   1:  PR[91,3] = PR[90,3] + 75.576;
   1:L PR[91] R[100]mm/sec CNT100;
   1:  PR[91,1] = PR[90,1] + -58.214;
   1:  PR[91,2] = PR[90,2] + 18.783;
   1:  PR[91,3] = PR[90,3] + 75.587;
   1:L PR[91] R[100]mm/sec CNT100;
   1:  PR[91] = PR[90];
   1:  PR[91,1] = PR[90,1] + -61.321;
   1:  PR[91,2] = PR[90,2] + 16.488;
   1:  PR[91,3] = PR[90,3] + 76.895;
   1:L PR[91] R[100]mm/sec CNT100;
   1:  PR[91,1] = PR[90,1] + -61.751;
   1:  PR[91,2] = PR[90,2] + 16.148;
   1:  PR[91,3] = PR[90,3] + 75.611;
   1:L PR[91] R[100]mm/sec CNT100;
   1:  PR[91,1] = PR[90,1] + -63.245;
   1:  PR[91,2] = PR[90,2] + 14.908;
   1:  PR[91,3] = PR[90,3] + 75.613;
   1:L PR[91] R[100]mm/sec CNT100;
   1:  PR[91,1] = PR[90,1] + -65.760;
   1:  PR[91,2] = PR[90,2] + 12.618;
   1:  PR[91,3] = PR[90,3] + 75.621;
   1:L PR[91] R[100]mm/sec CNT100;
   1:  PR[91,1] = PR[90,1] + -68.800;
   1:  PR[91,2] = PR[90,2] + 8.357;
   1:  PR[91,3] = PR[90,3] + 75.634;
   1:L PR[91] R[100]mm/sec CNT100;
   1:  PR[91,1] = PR[90,1] + -70.612;
   1:  PR[91,2] = PR[90,2] + 3.865;
   1:  PR[91,3] = PR[90,3] + 75.654;
   1:L PR[91] R[100]mm/sec CNT100;
   1:  PR[91,1] = PR[90,1] + -70.919;
   1:  PR[91,2] = PR[90,2] + 1.527;
   1:  PR[91,3] = PR[90,3] + 75.672;
   1:L PR[91] R[100]mm/sec CNT100;
   1:  PR[91,1] = PR[90,1] + -71.311;
   1:  PR[91,2] = PR[90,2] + -0.699;
   1:  PR[91,3] = PR[90,3] + 75.682;
   1:L PR[91] R[100]mm/sec CNT100;
   1:  PR[91,1] = PR[90,1] + -71.180;
   1:  PR[91,2] = PR[90,2] + -1.329;
   1:  PR[91,3] = PR[90,3] + 75.690;
   1:L PR[91] R[100]mm/sec CNT100;
   1:  PR[91,1] = PR[90,1] + -70.648;
   1:  PR[91,2] = PR[90,2] + -5.468;
   1:  PR[91,3] = PR[90,3] + 75.693;
   1:L PR[91] R[100]mm/sec CNT100;
   1:  PR[91,1] = PR[90,1] + -68.806;
   1:  PR[91,2] = PR[90,2] + -10.057;
   1:  PR[91,3] = PR[90,3] + 75.709;
   1:L PR[91] R[100]mm/sec CNT100;
   1:  PR[91,1] = PR[90,1] + -68.274;
   1:  PR[91,2] = PR[90,2] + -10.806;
   1:  PR[91,3] = PR[90,3] + 75.728;
   1:L PR[91] R[100]mm/sec CNT100;
   1:  PR[91,1] = PR[90,1] + -65.619;
   1:  PR[91,2] = PR[90,2] + -14.212;
   1:  PR[91,3] = PR[90,3] + 75.731;
   1:L PR[91] R[100]mm/sec CNT100;
   1:  PR[91,1] = PR[90,1] + -64.867;
   1:  PR[91,2] = PR[90,2] + -14.891;
   1:  PR[91,3] = PR[90,3] + 75.748;
   1:L PR[91] R[100]mm/sec CNT100;
   1:  PR[91,1] = PR[90,1] + -61.355;
   1:  PR[91,2] = PR[90,2] + -17.818;
   1:  PR[91,3] = PR[90,3] + 75.752;
   1:L PR[91] R[100]mm/sec CNT100;
   1:  PR[91,1] = PR[90,1] + -58.279;
   1:  PR[91,2] = PR[90,2] + -19.704;
   1:  PR[91,3] = PR[90,3] + 75.769;
   1:L PR[91] R[100]mm/sec CNT100;
   1:  PR[91,1] = PR[90,1] + -56.388;
   1:  PR[91,2] = PR[90,2] + -20.757;
   1:  PR[91,3] = PR[90,3] + 75.783;
   1:L PR[91] R[100]mm/sec CNT100;
   1:  PR[91,1] = PR[90,1] + -52.808;
   1:  PR[91,2] = PR[90,2] + -22.216;
   1:  PR[91,3] = PR[90,3] + 75.791;
   1:L PR[91] R[100]mm/sec CNT100;
   1:  PR[91,1] = PR[90,1] + -51.042;
   1:  PR[91,2] = PR[90,2] + -22.876;
   1:  PR[91,3] = PR[90,3] + 75.806;
   1:L PR[91] R[100]mm/sec CNT100;
   1:  PR[91,1] = PR[90,1] + -50.028;
   1:  PR[91,2] = PR[90,2] + -23.222;
   1:  PR[91,3] = PR[90,3] + 75.813;
   1:L PR[91] R[100]mm/sec CNT100;
   1:  PR[91,1] = PR[90,1] + -45.759;
   1:  PR[91,2] = PR[90,2] + -24.206;
   1:  PR[91,3] = PR[90,3] + 75.817;
   1:L PR[91] R[100]mm/sec CNT100;
   1:  PR[91,1] = PR[90,1] + -40.300;
   1:  PR[91,2] = PR[90,2] + -25.279;
   1:  PR[91,3] = PR[90,3] + 75.834;
   1:L PR[91] R[100]mm/sec CNT100;
   1:  PR[91,1] = PR[90,1] + -33.010;
   1:  PR[91,2] = PR[90,2] + -25.861;
   1:  PR[91,3] = PR[90,3] + 75.855;
   1:L PR[91] R[100]mm/sec CNT100;
   1:  PR[91,1] = PR[90,1] + -26.617;
   1:  PR[91,2] = PR[90,2] + -26.061;
   1:  PR[91,3] = PR[90,3] + 75.884;
   1:L PR[91] R[100]mm/sec CNT100;
   1:  PR[91,1] = PR[90,1] + -16.860;
   1:  PR[91,2] = PR[90,2] + -25.700;
   1:  PR[91,3] = PR[90,3] + 75.908;
   1:L PR[91] R[100]mm/sec CNT100;
   1:  PR[91,1] = PR[90,1] + -16.514;
   1:  PR[91,2] = PR[90,2] + -25.675;
   1:  PR[91,3] = PR[90,3] + 75.945;
   1:L PR[91] R[100]mm/sec CNT100;
   1:  PR[91,1] = PR[90,1] + -11.759;
   1:  PR[91,2] = PR[90,2] + -25.135;
   1:  PR[91,3] = PR[90,3] + 75.947;
   1:L PR[91] R[100]mm/sec CNT100;
   1:  PR[91,1] = PR[90,1] + -10.834;
   1:  PR[91,2] = PR[90,2] + -25.105;
   1:  PR[91,3] = PR[90,3] + 75.965;
   1:L PR[91] R[100]mm/sec CNT100;
   1:  PR[91,1] = PR[90,1] + -9.602;
   1:  PR[91,2] = PR[90,2] + -24.937;
   1:  PR[91,3] = PR[90,3] + 75.969;
   1:L PR[91] R[100]mm/sec CNT100;
   1:  PR[91,1] = PR[90,1] + -7.923;
   1:  PR[91,2] = PR[90,2] + -25.330;
   1:  PR[91,3] = PR[90,3] + 75.973;
   1:L PR[91] R[100]mm/sec CNT100;
   1:  PR[91,1] = PR[90,1] + -3.823;
   1:  PR[91,2] = PR[90,2] + -25.725;
   1:  PR[91,3] = PR[90,3] + 75.980;
   1:L PR[91] R[100]mm/sec CNT100;
   1:  PR[91,1] = PR[90,1] + -1.693;
   1:  PR[91,2] = PR[90,2] + -25.951;
   1:  PR[91,3] = PR[90,3] + 75.996;
   1:L PR[91] R[100]mm/sec CNT100;
   1:  PR[91,1] = PR[90,1] + -0.935;
   1:  PR[91,2] = PR[90,2] + -25.962;
   1:  PR[91,3] = PR[90,3] + 76.004;
   1:L PR[91] R[100]mm/sec CNT100;
   1:  PR[91,1] = PR[90,1] + 4.101;
   1:  PR[91,2] = PR[90,2] + -25.614;
   1:  PR[91,3] = PR[90,3] + 76.007;
   1:L PR[91] R[100]mm/sec CNT100;
   1:  PR[91,1] = PR[90,1] + 6.267;
   1:  PR[91,2] = PR[90,2] + -25.357;
   1:  PR[91,3] = PR[90,3] + 76.026;
   1:L PR[91] R[100]mm/sec CNT100;
   1:  PR[91,1] = PR[90,1] + 6.639;
   1:  PR[91,2] = PR[90,2] + -25.282;
   1:  PR[91,3] = PR[90,3] + 76.035;
   1:L PR[91] R[100]mm/sec CNT100;
   1:  PR[91,1] = PR[90,1] + 9.233;
   1:  PR[91,2] = PR[90,2] + -24.616;
   1:  PR[91,3] = PR[90,3] + 76.036;
   1:L PR[91] R[100]mm/sec CNT100;
   1:  PR[91,1] = PR[90,1] + 10.669;
   1:  PR[91,2] = PR[90,2] + -25.276;
   1:  PR[91,3] = PR[90,3] + 76.046;
   1:L PR[91] R[100]mm/sec CNT100;
   1:  PR[91,1] = PR[90,1] + 11.562;
   1:  PR[91,2] = PR[90,2] + -25.519;
   1:  PR[91,3] = PR[90,3] + 76.052;
   1:L PR[91] R[100]mm/sec CNT100;
   1:  PR[91,1] = PR[90,1] + 16.871;
   1:  PR[91,2] = PR[90,2] + -26.664;
   1:  PR[91,3] = PR[90,3] + 76.056;
   1:L PR[91] R[100]mm/sec CNT100;
   1:  PR[91,1] = PR[90,1] + 18.179;
   1:  PR[91,2] = PR[90,2] + -26.717;
   1:  PR[91,3] = PR[90,3] + 76.077;
   1:L PR[91] R[100]mm/sec CNT100;
   1:  PR[91,1] = PR[90,1] + 23.121;
   1:  PR[91,2] = PR[90,2] + -26.558;
   1:  PR[91,3] = PR[90,3] + 76.082;
   1:L PR[91] R[100]mm/sec CNT100;
   1:  PR[91,1] = PR[90,1] + 25.230;
   1:  PR[91,2] = PR[90,2] + -26.240;
   1:  PR[91,3] = PR[90,3] + 76.101;
   1:L PR[91] R[100]mm/sec CNT100;
   1:  PR[91,1] = PR[90,1] + 28.911;
   1:  PR[91,2] = PR[90,2] + -27.201;
   1:  PR[91,3] = PR[90,3] + 76.109;
   1:L PR[91] R[100]mm/sec CNT100;
   1:  PR[91,1] = PR[90,1] + 30.544;
   1:  PR[91,2] = PR[90,2] + -27.575;
   1:  PR[91,3] = PR[90,3] + 76.124;
   1:L PR[91] R[100]mm/sec CNT100;
   1:  PR[91,1] = PR[90,1] + 35.732;
   1:  PR[91,2] = PR[90,2] + -27.991;
   1:  PR[91,3] = PR[90,3] + 76.130;
   1:L PR[91] R[100]mm/sec CNT100;
   1:  PR[91,1] = PR[90,1] + 36.008;
   1:  PR[91,2] = PR[90,2] + -27.986;
   1:  PR[91,3] = PR[90,3] + 76.150;
   1:L PR[91] R[100]mm/sec CNT100;
   1:  PR[91,1] = PR[90,1] + 40.601;
   1:  PR[91,2] = PR[90,2] + -27.632;
   1:  PR[91,3] = PR[90,3] + 76.151;
   1:L PR[91] R[100]mm/sec CNT100;
   1:  PR[91,1] = PR[90,1] + 43.395;
   1:  PR[91,2] = PR[90,2] + -27.151;
   1:  PR[91,3] = PR[90,3] + 76.169;
   1:L PR[91] R[100]mm/sec CNT100;
   1:  PR[91,1] = PR[90,1] + 44.903;
   1:  PR[91,2] = PR[90,2] + -26.790;
   1:  PR[91,3] = PR[90,3] + 76.180;
   1:L PR[91] R[100]mm/sec CNT100;
   1:  PR[91,1] = PR[90,1] + 47.079;
   1:  PR[91,2] = PR[90,2] + -26.059;
   1:  PR[91,3] = PR[90,3] + 76.186;
   1:L PR[91] R[100]mm/sec CNT100;
   1:  PR[91,1] = PR[90,1] + 49.432;
   1:  PR[91,2] = PR[90,2] + -25.424;
   1:  PR[91,3] = PR[90,3] + 76.194;
   1:L PR[91] R[100]mm/sec CNT100;
   1:  PR[91,1] = PR[90,1] + 51.453;
   1:  PR[91,2] = PR[90,2] + -24.639;
   1:  PR[91,3] = PR[90,3] + 76.204;
   1:L PR[91] R[100]mm/sec CNT100;
   1:  PR[91,1] = PR[90,1] + 53.638;
   1:  PR[91,2] = PR[90,2] + -23.715;
   1:  PR[91,3] = PR[90,3] + 76.212;
   1:L PR[91] R[100]mm/sec CNT100;
   1:  PR[91,1] = PR[90,1] + 55.403;
   1:  PR[91,2] = PR[90,2] + -22.742;
   1:  PR[91,3] = PR[90,3] + 76.221;
   1:L PR[91] R[100]mm/sec CNT100;
   1:  PR[91,1] = PR[90,1] + 57.643;
   1:  PR[91,2] = PR[90,2] + -21.692;
   1:  PR[91,3] = PR[90,3] + 76.229;
   1:L PR[91] R[100]mm/sec CNT100;
   1:  PR[91,1] = PR[90,1] + 61.600;
   1:  PR[91,2] = PR[90,2] + -19.230;
   1:  PR[91,3] = PR[90,3] + 76.238;
   1:L PR[91] R[100]mm/sec CNT100;
   1:  PR[91,1] = PR[90,1] + 65.239;
   1:  PR[91,2] = PR[90,2] + -16.034;
   1:  PR[91,3] = PR[90,3] + 76.256;
   1:L PR[91] R[100]mm/sec CNT100;
   1:  PR[91,1] = PR[90,1] + 66.422;
   1:  PR[91,2] = PR[90,2] + -14.530;
   1:  PR[91,3] = PR[90,3] + 76.275;
   1:L PR[91] R[100]mm/sec CNT100;
   1:  PR[91,1] = PR[90,1] + 68.582;
   1:  PR[91,2] = PR[90,2] + -11.849;
   1:  PR[91,3] = PR[90,3] + 76.282;
   1:L PR[91] R[100]mm/sec CNT100;
   1:  PR[91,1] = PR[90,1] + 69.577;
   1:  PR[91,2] = PR[90,2] + -10.060;
   1:  PR[91,3] = PR[90,3] + 76.295;
   1:L PR[91] R[100]mm/sec CNT100;
   1:  PR[91,1] = PR[90,1] + 70.915;
   1:  PR[91,2] = PR[90,2] + -7.005;
   1:  PR[91,3] = PR[90,3] + 76.303;
   1:L PR[91] R[100]mm/sec CNT100;
   1:  PR[91,1] = PR[90,1] + 71.354;
   1:  PR[91,2] = PR[90,2] + -5.640;
   1:  PR[91,3] = PR[90,3] + 76.316;
   1:L PR[91] R[100]mm/sec CNT100;
   1:  PR[91,1] = PR[90,1] + 71.890;
   1:  PR[91,2] = PR[90,2] + -1.894;
   1:  PR[91,3] = PR[90,3] + 76.321;
   1:L PR[91] R[100]mm/sec CNT100;
   1:  PR[91,1] = PR[90,1] + 72.009;
   1:  PR[91,2] = PR[90,2] + -0.768;
   1:  PR[91,3] = PR[90,3] + 76.336;
   1:L PR[91] R[100]mm/sec CNT100;
   1:  PR[91,1] = PR[90,1] + 71.482;
   1:  PR[91,2] = PR[90,2] + 2.880;
   1:  PR[91,3] = PR[90,3] + 76.340;
   1:L PR[91] R[100]mm/sec CNT100;
   1:  PR[91,1] = PR[90,1] + 71.343;
   1:  PR[91,2] = PR[90,2] + 4.216;
   1:  PR[91,3] = PR[90,3] + 76.354;
   1:L PR[91] R[100]mm/sec CNT100;
   1:  PR[91,1] = PR[90,1] + 70.915;
   1:  PR[91,2] = PR[90,2] + 5.544;
   1:  PR[91,3] = PR[90,3] + 76.359;
   1:L PR[91] R[100]mm/sec CNT100;
   1:  PR[91,1] = PR[90,1] + 69.579;
   1:  PR[91,2] = PR[90,2] + 8.598;
   1:  PR[91,3] = PR[90,3] + 76.365;
   1:L PR[91] R[100]mm/sec CNT100;
   1:  PR[91,1] = PR[90,1] + 68.577;
   1:  PR[91,2] = PR[90,2] + 10.401;
   1:  PR[91,3] = PR[90,3] + 76.378;
   1:L PR[91] R[100]mm/sec CNT100;
   1:  PR[91,1] = PR[90,1] + 67.100;
   1:  PR[91,2] = PR[90,2] + 12.290;
   1:  PR[91,3] = PR[90,3] + 76.386;
   1:L PR[91] R[100]mm/sec CNT100;
   1:  PR[91,1] = PR[90,1] + 65.254;
   1:  PR[91,2] = PR[90,2] + 14.562;
   1:  PR[91,3] = PR[90,3] + 76.395;
   1:L PR[91] R[100]mm/sec CNT100;
   1:  PR[91,1] = PR[90,1] + 61.600;
   1:  PR[91,2] = PR[90,2] + 17.771;
   1:  PR[91,3] = PR[90,3] + 76.406;
   1:L PR[91] R[100]mm/sec CNT100;
   1:  PR[91,1] = PR[90,1] + 57.643;
   1:  PR[91,2] = PR[90,2] + 20.234;
   1:  PR[91,3] = PR[90,3] + 76.425;
   1:L PR[91] R[100]mm/sec CNT100;
   1:  PR[91,1] = PR[90,1] + 55.403;
   1:  PR[91,2] = PR[90,2] + 21.284;
   1:  PR[91,3] = PR[90,3] + 76.442;
   1:L PR[91] R[100]mm/sec CNT100;
   1:  PR[91,1] = PR[90,1] + 53.638;
   1:  PR[91,2] = PR[90,2] + 22.256;
   1:  PR[91,3] = PR[90,3] + 76.452;
   1:L PR[91] R[100]mm/sec CNT100;
   1:  PR[91,1] = PR[90,1] + 51.453;
   1:  PR[91,2] = PR[90,2] + 23.180;
   1:  PR[91,3] = PR[90,3] + 76.460;
   1:L PR[91] R[100]mm/sec CNT100;
   1:  PR[91,1] = PR[90,1] + 49.432;
   1:  PR[91,2] = PR[90,2] + 23.965;
   1:  PR[91,3] = PR[90,3] + 76.469;
   1:L PR[91] R[100]mm/sec CNT100;
   1:  PR[91,1] = PR[90,1] + 47.079;
   1:  PR[91,2] = PR[90,2] + 24.601;
   1:  PR[91,3] = PR[90,3] + 76.477;
   1:L PR[91] R[100]mm/sec CNT100;
   1:  PR[91,1] = PR[90,1] + 44.903;
   1:  PR[91,2] = PR[90,2] + 25.331;
   1:  PR[91,3] = PR[90,3] + 76.486;
   1:L PR[91] R[100]mm/sec CNT100;
   1:  PR[91,1] = PR[90,1] + 43.395;
   1:  PR[91,2] = PR[90,2] + 25.692;
   1:  PR[91,3] = PR[90,3] + 76.495;
   1:L PR[91] R[100]mm/sec CNT100;
   1:  PR[91,1] = PR[90,1] + 40.601;
   1:  PR[91,2] = PR[90,2] + 26.173;
   1:  PR[91,3] = PR[90,3] + 76.501;
   1:L PR[91] R[100]mm/sec CNT100;
   1:  PR[91,1] = PR[90,1] + 36.008;
   1:  PR[91,2] = PR[90,2] + 26.528;
   1:  PR[91,3] = PR[90,3] + 76.512;
   1:L PR[91] R[100]mm/sec CNT100;
   1:  PR[91,1] = PR[90,1] + 35.732;
   1:  PR[91,2] = PR[90,2] + 26.532;
   1:  PR[91,3] = PR[90,3] + 76.530;
   1:L PR[91] R[100]mm/sec CNT100;
   1:  PR[91,1] = PR[90,1] + 30.544;
   1:  PR[91,2] = PR[90,2] + 26.116;
   1:  PR[91,3] = PR[90,3] + 76.531;
   1:L PR[91] R[100]mm/sec CNT100;
   1:  PR[91,1] = PR[90,1] + 28.911;
   1:  PR[91,2] = PR[90,2] + 25.742;
   1:  PR[91,3] = PR[90,3] + 76.551;
   1:L PR[91] R[100]mm/sec CNT100;
   1:  PR[91,1] = PR[90,1] + 25.230;
   1:  PR[91,2] = PR[90,2] + 24.781;
   1:  PR[91,3] = PR[90,3] + 76.557;
   1:L PR[91] R[100]mm/sec CNT100;
   1:  PR[91,1] = PR[90,1] + 23.121;
   1:  PR[91,2] = PR[90,2] + 25.099;
   1:  PR[91,3] = PR[90,3] + 76.572;
   1:L PR[91] R[100]mm/sec CNT100;
   1:  PR[91,1] = PR[90,1] + 18.179;
   1:  PR[91,2] = PR[90,2] + 25.258;
   1:  PR[91,3] = PR[90,3] + 76.580;
   1:L PR[91] R[100]mm/sec CNT100;
   1:  PR[91,1] = PR[90,1] + 16.870;
   1:  PR[91,2] = PR[90,2] + 25.205;
   1:  PR[91,3] = PR[90,3] + 76.599;
   1:L PR[91] R[100]mm/sec CNT100;
   1:  PR[91,1] = PR[90,1] + 11.562;
   1:  PR[91,2] = PR[90,2] + 24.060;
   1:  PR[91,3] = PR[90,3] + 76.604;
   1:L PR[91] R[100]mm/sec CNT100;
   1:  PR[91,1] = PR[90,1] + 10.668;
   1:  PR[91,2] = PR[90,2] + 23.817;
   1:  PR[91,3] = PR[90,3] + 76.625;
   1:L PR[91] R[100]mm/sec CNT100;
   1:  PR[91,1] = PR[90,1] + 9.232;
   1:  PR[91,2] = PR[90,2] + 23.158;
   1:  PR[91,3] = PR[90,3] + 76.628;
   1:L PR[91] R[100]mm/sec CNT100;
   1:  PR[91,1] = PR[90,1] + 6.658;
   1:  PR[91,2] = PR[90,2] + 23.820;
   1:  PR[91,3] = PR[90,3] + 76.634;
   1:L PR[91] R[100]mm/sec CNT100;
   1:  PR[91,1] = PR[90,1] + 6.292;
   1:  PR[91,2] = PR[90,2] + 23.894;
   1:  PR[91,3] = PR[90,3] + 76.644;
   1:L PR[91] R[100]mm/sec CNT100;
   1:  PR[91,1] = PR[90,1] + 4.125;
   1:  PR[91,2] = PR[90,2] + 24.151;
   1:  PR[91,3] = PR[90,3] + 76.646;
   1:L PR[91] R[100]mm/sec CNT100;
   1:  PR[91,1] = PR[90,1] + -0.919;
   1:  PR[91,2] = PR[90,2] + 24.504;
   1:  PR[91,3] = PR[90,3] + 76.654;
   1:L PR[91] R[100]mm/sec CNT100;
   1:  PR[91,1] = PR[90,1] + -1.502;
   1:  PR[91,2] = PR[90,2] + 24.503;
   1:  PR[91,3] = PR[90,3] + 76.674;
   1:L PR[91] R[100]mm/sec CNT100;
   1:  PR[91,1] = PR[90,1] + -7.921;
   1:  PR[91,2] = PR[90,2] + 23.871;
   1:  PR[91,3] = PR[90,3] + 76.676;
   1:L PR[91] R[100]mm/sec CNT100;
   1:  PR[91,1] = PR[90,1] + -9.601;
   1:  PR[91,2] = PR[90,2] + 23.477;
   1:  PR[91,3] = PR[90,3] + 76.701;
   1:L PR[91] R[100]mm/sec CNT100;
   1:  PR[91,1] = PR[90,1] + -10.909;
   1:  PR[91,2] = PR[90,2] + 23.656;
   1:  PR[91,3] = PR[90,3] + 76.707;
   1:L PR[91] R[100]mm/sec CNT100;
   1:  PR[91,1] = PR[90,1] + -13.256;
   1:  PR[91,2] = PR[90,2] + 23.913;
   1:  PR[91,3] = PR[90,3] + 76.712;
   1:L PR[91] R[100]mm/sec CNT100;
   1:  PR[91,1] = PR[90,1] + -16.734;
   1:  PR[91,2] = PR[90,2] + 24.232;
   1:  PR[91,3] = PR[90,3] + 76.721;
   1:L PR[91] R[100]mm/sec CNT100;
   1:  PR[91,1] = PR[90,1] + -26.619;
   1:  PR[91,2] = PR[90,2] + 24.602;
   1:  PR[91,3] = PR[90,3] + 76.735;
   1:L PR[91] R[100]mm/sec CNT100;
   1:  PR[91,1] = PR[90,1] + -32.992;
   1:  PR[91,2] = PR[90,2] + 24.411;
   1:  PR[91,3] = PR[90,3] + 76.773;
   1:L PR[91] R[100]mm/sec CNT100;
   1:  PR[91,1] = PR[90,1] + -38.952;
   1:  PR[91,2] = PR[90,2] + 23.902;
   1:  PR[91,3] = PR[90,3] + 76.797;
   1:L PR[91] R[100]mm/sec CNT100;
   1:  PR[91,1] = PR[90,1] + -40.166;
   1:  PR[91,2] = PR[90,2] + 23.822;
   1:  PR[91,3] = PR[90,3] + 76.820;
   1:L PR[91] R[100]mm/sec CNT100;
   1:  PR[91,1] = PR[90,1] + -42.567;
   1:  PR[91,2] = PR[90,2] + 23.411;
   1:  PR[91,3] = PR[90,3] + 76.825;
   1:L PR[91] R[100]mm/sec CNT100;
   1:  PR[91,1] = PR[90,1] + -47.291;
   1:  PR[91,2] = PR[90,2] + 22.501;
   1:  PR[91,3] = PR[90,3] + 76.834;
   1:L PR[91] R[100]mm/sec CNT100;
   1:  PR[91,1] = PR[90,1] + -50.078;
   1:  PR[91,2] = PR[90,2] + 21.634;
   1:  PR[91,3] = PR[90,3] + 76.852;
   1:L PR[91] R[100]mm/sec CNT100;
   1:  PR[91,1] = PR[90,1] + -53.115;
   1:  PR[91,2] = PR[90,2] + 20.640;
   1:  PR[91,3] = PR[90,3] + 76.864;
   1:L PR[91] R[100]mm/sec CNT100;
   1:  PR[91,1] = PR[90,1] + -54.843;
   1:  PR[91,2] = PR[90,2] + 20.012;
   1:  PR[91,3] = PR[90,3] + 76.876;
   1:L PR[91] R[100]mm/sec CNT100;
   1:  PR[91,1] = PR[90,1] + -57.622;
   1:  PR[91,2] = PR[90,2] + 18.557;
   1:  PR[91,3] = PR[90,3] + 76.883;
   1:L PR[91] R[100]mm/sec CNT100;
   1:  PR[91] = PR[90];
   1:  PR[91,1] = PR[90,1] + -59.923;
   1:  PR[91,2] = PR[90,2] + 16.713;
   1:  PR[91,3] = PR[90,3] + 78.195;
   1:L PR[91] R[100]mm/sec CNT100;
   1:  PR[91,1] = PR[90,1] + -61.088;
   1:  PR[91,2] = PR[90,2] + 15.792;
   1:  PR[91,3] = PR[90,3] + 76.908;
   1:L PR[91] R[100]mm/sec CNT100;
   1:  PR[91,1] = PR[90,1] + -64.563;
   1:  PR[91,2] = PR[90,2] + 12.906;
   1:  PR[91,3] = PR[90,3] + 76.914;
   1:L PR[91] R[100]mm/sec CNT100;
   1:  PR[91,1] = PR[90,1] + -64.751;
   1:  PR[91,2] = PR[90,2] + 12.734;
   1:  PR[91,3] = PR[90,3] + 76.931;
   1:L PR[91] R[100]mm/sec CNT100;
   1:  PR[91,1] = PR[90,1] + -67.821;
   1:  PR[91,2] = PR[90,2] + 8.435;
   1:  PR[91,3] = PR[90,3] + 76.932;
   1:L PR[91] R[100]mm/sec CNT100;
   1:  PR[91,1] = PR[90,1] + -69.130;
   1:  PR[91,2] = PR[90,2] + 5.200;
   1:  PR[91,3] = PR[90,3] + 76.953;
   1:L PR[91] R[100]mm/sec CNT100;
   1:  PR[91,1] = PR[90,1] + -69.650;
   1:  PR[91,2] = PR[90,2] + 3.906;
   1:  PR[91,3] = PR[90,3] + 76.966;
   1:L PR[91] R[100]mm/sec CNT100;
   1:  PR[91,1] = PR[90,1] + -69.862;
   1:  PR[91,2] = PR[90,2] + 2.292;
   1:  PR[91,3] = PR[90,3] + 76.972;
   1:L PR[91] R[100]mm/sec CNT100;
   1:  PR[91,1] = PR[90,1] + -70.389;
   1:  PR[91,2] = PR[90,2] + -0.698;
   1:  PR[91,3] = PR[90,3] + 76.978;
   1:L PR[91] R[100]mm/sec CNT100;
   1:  PR[91,1] = PR[90,1] + -70.382;
   1:  PR[91,2] = PR[90,2] + -0.732;
   1:  PR[91,3] = PR[90,3] + 76.990;
   1:L PR[91] R[100]mm/sec CNT100;
   1:  PR[91,1] = PR[90,1] + -69.769;
   1:  PR[91,2] = PR[90,2] + -5.495;
   1:L PR[91] R[100]mm/sec CNT100;
   1:  PR[91,1] = PR[90,1] + -69.452;
   1:  PR[91,2] = PR[90,2] + -6.286;
   1:  PR[91,3] = PR[90,3] + 77.008;
   1:L PR[91] R[100]mm/sec CNT100;
   1:  PR[91,1] = PR[90,1] + -67.800;
   1:  PR[91,2] = PR[90,2] + -10.028;
   1:  PR[91,3] = PR[90,3] + 77.012;
   1:L PR[91] R[100]mm/sec CNT100;
   1:  PR[91,1] = PR[90,1] + -67.559;
   1:  PR[91,2] = PR[90,2] + -10.359;
   1:  PR[91,3] = PR[90,3] + 77.028;
   1:L PR[91] R[100]mm/sec CNT100;
   1:  PR[91,1] = PR[90,1] + -64.570;
   1:  PR[91,2] = PR[90,2] + -14.196;
   1:  PR[91,3] = PR[90,3] + 77.029;
   1:L PR[91] R[100]mm/sec CNT100;
   1:  PR[91,1] = PR[90,1] + -63.011;
   1:  PR[91,2] = PR[90,2] + -15.601;
   1:  PR[91,3] = PR[90,3] + 77.048;
   1:L PR[91] R[100]mm/sec CNT100;
   1:  PR[91,1] = PR[90,1] + -60.356;
   1:  PR[91,2] = PR[90,2] + -17.814;
   1:  PR[91,3] = PR[90,3] + 77.056;
   1:L PR[91] R[100]mm/sec CNT100;
   1:  PR[91,1] = PR[90,1] + -56.217;
   1:  PR[91,2] = PR[90,2] + -20.352;
   1:  PR[91,3] = PR[90,3] + 77.070;
   1:L PR[91] R[100]mm/sec CNT100;
   1:  PR[91,1] = PR[90,1] + -55.448;
   1:  PR[91,2] = PR[90,2] + -20.781;
   1:  PR[91,3] = PR[90,3] + 77.088;
   1:L PR[91] R[100]mm/sec CNT100;
   1:  PR[91,1] = PR[90,1] + -53.919;
   1:  PR[91,2] = PR[90,2] + -21.404;
   1:  PR[91,3] = PR[90,3] + 77.092;
   1:L PR[91] R[100]mm/sec CNT100;
   1:  PR[91,1] = PR[90,1] + -50.274;
   1:  PR[91,2] = PR[90,2] + -22.767;
   1:  PR[91,3] = PR[90,3] + 77.098;
   1:L PR[91] R[100]mm/sec CNT100;
   1:  PR[91,1] = PR[90,1] + -48.085;
   1:  PR[91,2] = PR[90,2] + -23.514;
   1:  PR[91,3] = PR[90,3] + 77.113;
   1:L PR[91] R[100]mm/sec CNT100;
   1:  PR[91,1] = PR[90,1] + -45.017;
   1:  PR[91,2] = PR[90,2] + -24.221;
   1:  PR[91,3] = PR[90,3] + 77.122;
   1:L PR[91] R[100]mm/sec CNT100;
   1:  PR[91,1] = PR[90,1] + -40.786;
   1:  PR[91,2] = PR[90,2] + -25.052;
   1:  PR[91,3] = PR[90,3] + 77.134;
   1:L PR[91] R[100]mm/sec CNT100;
   1:  PR[91,1] = PR[90,1] + -38.694;
   1:  PR[91,2] = PR[90,2] + -25.441;
   1:  PR[91,3] = PR[90,3] + 77.151;
   1:L PR[91] R[100]mm/sec CNT100;
   1:  PR[91,1] = PR[90,1] + -36.027;
   1:  PR[91,2] = PR[90,2] + -25.726;
   1:  PR[91,3] = PR[90,3] + 77.159;
   1:L PR[91] R[100]mm/sec CNT100;
   1:  PR[91,1] = PR[90,1] + -31.850;
   1:  PR[91,2] = PR[90,2] + -26.059;
   1:  PR[91,3] = PR[90,3] + 77.170;
   1:L PR[91] R[100]mm/sec CNT100;
   1:  PR[91,1] = PR[90,1] + -23.988;
   1:  PR[91,2] = PR[90,2] + -26.313;
   1:  PR[91,3] = PR[90,3] + 77.186;
   1:L PR[91] R[100]mm/sec CNT100;
   1:  PR[91,1] = PR[90,1] + -14.147;
   1:  PR[91,2] = PR[90,2] + -25.955;
   1:  PR[91,3] = PR[90,3] + 77.217;
   1:L PR[91] R[100]mm/sec CNT100;
   1:  PR[91,1] = PR[90,1] + -13.688;
   1:  PR[91,2] = PR[90,2] + -25.922;
   1:  PR[91,3] = PR[90,3] + 77.255;
   1:L PR[91] R[100]mm/sec CNT100;
   1:  PR[91,1] = PR[90,1] + -9.685;
   1:  PR[91,2] = PR[90,2] + -25.467;
   1:  PR[91,3] = PR[90,3] + 77.257;
   1:L PR[91] R[100]mm/sec CNT100;
   1:  PR[91,1] = PR[90,1] + -8.709;
   1:  PR[91,2] = PR[90,2] + -25.441;
   1:  PR[91,3] = PR[90,3] + 77.272;
   1:L PR[91] R[100]mm/sec CNT100;
   1:  PR[91,1] = PR[90,1] + -7.981;
   1:  PR[91,2] = PR[90,2] + -25.351;
   1:  PR[91,3] = PR[90,3] + 77.276;
   1:L PR[91] R[100]mm/sec CNT100;
   1:  PR[91,1] = PR[90,1] + -7.226;
   1:  PR[91,2] = PR[90,2] + -25.528;
   1:  PR[91,3] = PR[90,3] + 77.279;
   1:L PR[91] R[100]mm/sec CNT100;
   1:  PR[91,1] = PR[90,1] + -5.779;
   1:  PR[91,2] = PR[90,2] + -25.667;
   1:  PR[91,3] = PR[90,3] + 77.282;
   1:L PR[91] R[100]mm/sec CNT100;
   1:  PR[91,1] = PR[90,1] + -1.148;
   1:  PR[91,2] = PR[90,2] + -26.158;
   1:  PR[91,3] = PR[90,3] + 77.287;
   1:L PR[91] R[100]mm/sec CNT100;
   1:  PR[91,1] = PR[90,1] + -0.859;
   1:  PR[91,2] = PR[90,2] + -26.177;
   1:  PR[91,3] = PR[90,3] + 77.306;
   1:L PR[91] R[100]mm/sec CNT100;
   1:  PR[91,1] = PR[90,1] + 0.581;
   1:  PR[91,2] = PR[90,2] + -26.180;
   1:  PR[91,3] = PR[90,3] + 77.307;
   1:L PR[91] R[100]mm/sec CNT100;
   1:  PR[91,1] = PR[90,1] + 4.613;
   1:  PR[91,2] = PR[90,2] + -25.901;
   1:  PR[91,3] = PR[90,3] + 77.312;
   1:L PR[91] R[100]mm/sec CNT100;
   1:  PR[91,1] = PR[90,1] + 7.461;
   1:  PR[91,2] = PR[90,2] + -25.564;
   1:  PR[91,3] = PR[90,3] + 77.328;
   1:L PR[91] R[100]mm/sec CNT100;
   1:  PR[91,1] = PR[90,1] + 7.983;
   1:  PR[91,2] = PR[90,2] + -25.458;
   1:  PR[91,3] = PR[90,3] + 77.339;
   1:L PR[91] R[100]mm/sec CNT100;
   1:  PR[91,1] = PR[90,1] + 9.579;
   1:  PR[91,2] = PR[90,2] + -25.048;
   1:  PR[91,3] = PR[90,3] + 77.341;
   1:L PR[91] R[100]mm/sec CNT100;
   1:  PR[91,1] = PR[90,1] + 10.535;
   1:  PR[91,2] = PR[90,2] + -25.487;
   1:  PR[91,3] = PR[90,3] + 77.347;
   1:L PR[91] R[100]mm/sec CNT100;
   1:  PR[91,1] = PR[90,1] + 10.865;
   1:  PR[91,2] = PR[90,2] + -25.577;
   1:  PR[91,3] = PR[90,3] + 77.352;
   1:L PR[91] R[100]mm/sec CNT100;
   1:  PR[91,1] = PR[90,1] + 16.833;
   1:  PR[91,2] = PR[90,2] + -26.865;
   1:  PR[91,3] = PR[90,3] + 77.353;
   1:L PR[91] R[100]mm/sec CNT100;
   1:  PR[91,1] = PR[90,1] + 17.573;
   1:  PR[91,2] = PR[90,2] + -26.895;
   1:  PR[91,3] = PR[90,3] + 77.377;
   1:L PR[91] R[100]mm/sec CNT100;
   1:  PR[91,1] = PR[90,1] + 23.172;
   1:  PR[91,2] = PR[90,2] + -26.714;
   1:  PR[91,3] = PR[90,3] + 77.379;
   1:L PR[91] R[100]mm/sec CNT100;
   1:  PR[91,1] = PR[90,1] + 24.763;
   1:  PR[91,2] = PR[90,2] + -26.476;
   1:  PR[91,3] = PR[90,3] + 77.401;
   1:L PR[91] R[100]mm/sec CNT100;
   1:  PR[91,1] = PR[90,1] + 27.460;
   1:  PR[91,2] = PR[90,2] + -27.180;
   1:  PR[91,3] = PR[90,3] + 77.407;
   1:L PR[91] R[100]mm/sec CNT100;
   1:  PR[91,1] = PR[90,1] + 30.172;
   1:  PR[91,2] = PR[90,2] + -27.801;
   1:  PR[91,3] = PR[90,3] + 77.418;
   1:L PR[91] R[100]mm/sec CNT100;
   1:  PR[91,1] = PR[90,1] + 34.661;
   1:  PR[91,2] = PR[90,2] + -28.160;
   1:  PR[91,3] = PR[90,3] + 77.429;
   1:L PR[91] R[100]mm/sec CNT100;
   1:  PR[91,1] = PR[90,1] + 35.284;
   1:  PR[91,2] = PR[90,2] + -28.195;
   1:  PR[91,3] = PR[90,3] + 77.446;
   1:L PR[91] R[100]mm/sec CNT100;
   1:  PR[91,1] = PR[90,1] + 36.831;
   1:  PR[91,2] = PR[90,2] + -28.047;
   1:  PR[91,3] = PR[90,3] + 77.449;
   1:L PR[91] R[100]mm/sec CNT100;
   1:  PR[91,1] = PR[90,1] + 40.358;
   1:  PR[91,2] = PR[90,2] + -27.775;
   1:  PR[91,3] = PR[90,3] + 77.455;
   1:L PR[91] R[100]mm/sec CNT100;
   1:  PR[91,1] = PR[90,1] + 41.931;
   1:  PR[91,2] = PR[90,2] + -27.504;
   1:  PR[91,3] = PR[90,3] + 77.469;
   1:L PR[91] R[100]mm/sec CNT100;
   1:  PR[91,1] = PR[90,1] + 44.773;
   1:  PR[91,2] = PR[90,2] + -26.824;
   1:  PR[91,3] = PR[90,3] + 77.475;
   1:L PR[91] R[100]mm/sec CNT100;
   1:  PR[91,1] = PR[90,1] + 48.715;
   1:  PR[91,2] = PR[90,2] + -25.508;
   1:  PR[91,3] = PR[90,3] + 77.486;
   1:L PR[91] R[100]mm/sec CNT100;
   1:  PR[91,1] = PR[90,1] + 53.139;
   1:  PR[91,2] = PR[90,2] + -23.641;
   1:  PR[91,3] = PR[90,3] + 77.502;
   1:L PR[91] R[100]mm/sec CNT100;
   1:  PR[91,1] = PR[90,1] + 56.598;
   1:  PR[91,2] = PR[90,2] + -21.735;
   1:  PR[91,3] = PR[90,3] + 77.521;
   1:L PR[91] R[100]mm/sec CNT100;
   1:  PR[91,1] = PR[90,1] + 56.791;
   1:  PR[91,2] = PR[90,2] + -21.644;
   1:  PR[91,3] = PR[90,3] + 77.536;
   1:L PR[91] R[100]mm/sec CNT100;
   1:  PR[91,1] = PR[90,1] + 60.697;
   1:  PR[91,2] = PR[90,2] + -19.149;
   1:  PR[91,3] = PR[90,3] + 77.537;
   1:L PR[91] R[100]mm/sec CNT100;
   1:  PR[91,1] = PR[90,1] + 62.864;
   1:  PR[91,2] = PR[90,2] + -17.319;
   1:  PR[91,3] = PR[90,3] + 77.555;
   1:L PR[91] R[100]mm/sec CNT100;
   1:  PR[91,1] = PR[90,1] + 64.236;
   1:  PR[91,2] = PR[90,2] + -16.111;
   1:  PR[91,3] = PR[90,3] + 77.566;
   1:L PR[91] R[100]mm/sec CNT100;
   1:  PR[91,1] = PR[90,1] + 67.448;
   1:  PR[91,2] = PR[90,2] + -12.111;
   1:  PR[91,3] = PR[90,3] + 77.573;
   1:L PR[91] R[100]mm/sec CNT100;
   1:  PR[91,1] = PR[90,1] + 68.762;
   1:  PR[91,2] = PR[90,2] + -9.747;
   1:  PR[91,3] = PR[90,3] + 77.593;
   1:L PR[91] R[100]mm/sec CNT100;
   1:  PR[91,1] = PR[90,1] + 69.760;
   1:  PR[91,2] = PR[90,2] + -7.466;
   1:  PR[91,3] = PR[90,3] + 77.603;
   1:L PR[91] R[100]mm/sec CNT100;
   1:  PR[91,1] = PR[90,1] + 70.405;
   1:  PR[91,2] = PR[90,2] + -5.465;
   1:  PR[91,3] = PR[90,3] + 77.613;
   1:L PR[91] R[100]mm/sec CNT100;
   1:  PR[91,1] = PR[90,1] + 70.823;
   1:  PR[91,2] = PR[90,2] + -2.539;
   1:  PR[91,3] = PR[90,3] + 77.621;
   1:L PR[91] R[100]mm/sec CNT100;
   1:  PR[91,1] = PR[90,1] + 71.010;
   1:  PR[91,2] = PR[90,2] + -0.768;
   1:  PR[91,3] = PR[90,3] + 77.633;
   1:L PR[91] R[100]mm/sec CNT100;
   1:  PR[91,1] = PR[90,1] + 70.594;
   1:  PR[91,2] = PR[90,2] + 2.114;
   1:  PR[91,3] = PR[90,3] + 77.640;
   1:L PR[91] R[100]mm/sec CNT100;
   1:  PR[91,1] = PR[90,1] + 70.394;
   1:  PR[91,2] = PR[90,2] + 4.041;
   1:  PR[91,3] = PR[90,3] + 77.651;
   1:L PR[91] R[100]mm/sec CNT100;
   1:  PR[91,1] = PR[90,1] + 69.761;
   1:  PR[91,2] = PR[90,2] + 6.006;
   1:  PR[91,3] = PR[90,3] + 77.658;
   1:L PR[91] R[100]mm/sec CNT100;
   1:  PR[91,1] = PR[90,1] + 68.763;
   1:  PR[91,2] = PR[90,2] + 8.286;
   1:  PR[91,3] = PR[90,3] + 77.666;
   1:L PR[91] R[100]mm/sec CNT100;
   1:  PR[91,1] = PR[90,1] + 67.443;
   1:  PR[91,2] = PR[90,2] + 10.661;
   1:  PR[91,3] = PR[90,3] + 77.676;
   1:L PR[91] R[100]mm/sec CNT100;
   1:  PR[91,1] = PR[90,1] + 66.473;
   1:  PR[91,2] = PR[90,2] + 11.902;
   1:  PR[91,3] = PR[90,3] + 77.687;
   1:L PR[91] R[100]mm/sec CNT100;
   1:  PR[91,1] = PR[90,1] + 64.242;
   1:  PR[91,2] = PR[90,2] + 14.647;
   1:  PR[91,3] = PR[90,3] + 77.693;
   1:L PR[91] R[100]mm/sec CNT100;
   1:  PR[91,1] = PR[90,1] + 62.864;
   1:  PR[91,2] = PR[90,2] + 15.860;
   1:  PR[91,3] = PR[90,3] + 77.706;
   1:L PR[91] R[100]mm/sec CNT100;
   1:  PR[91,1] = PR[90,1] + 60.697;
   1:  PR[91,2] = PR[90,2] + 17.690;
   1:  PR[91,3] = PR[90,3] + 77.714;
   1:L PR[91] R[100]mm/sec CNT100;
   1:  PR[91,1] = PR[90,1] + 56.791;
   1:  PR[91,2] = PR[90,2] + 20.186;
   1:  PR[91,3] = PR[90,3] + 77.725;
   1:L PR[91] R[100]mm/sec CNT100;
   1:  PR[91,1] = PR[90,1] + 56.598;
   1:  PR[91,2] = PR[90,2] + 20.276;
   1:  PR[91,3] = PR[90,3] + 77.743;
   1:L PR[91] R[100]mm/sec CNT100;
   1:  PR[91,1] = PR[90,1] + 53.139;
   1:  PR[91,2] = PR[90,2] + 22.182;
   1:L PR[91] R[100]mm/sec CNT100;
   1:  PR[91,1] = PR[90,1] + 48.715;
   1:  PR[91,2] = PR[90,2] + 24.049;
   1:  PR[91,3] = PR[90,3] + 77.759;
   1:L PR[91] R[100]mm/sec CNT100;
   1:  PR[91,1] = PR[90,1] + 44.774;
   1:  PR[91,2] = PR[90,2] + 25.365;
   1:  PR[91,3] = PR[90,3] + 77.777;
   1:L PR[91] R[100]mm/sec CNT100;
   1:  PR[91,1] = PR[90,1] + 41.931;
   1:  PR[91,2] = PR[90,2] + 26.046;
   1:  PR[91,3] = PR[90,3] + 77.793;
   1:L PR[91] R[100]mm/sec CNT100;
   1:  PR[91,1] = PR[90,1] + 40.358;
   1:  PR[91,2] = PR[90,2] + 26.316;
   1:  PR[91,3] = PR[90,3] + 77.805;
   1:L PR[91] R[100]mm/sec CNT100;
   1:  PR[91,1] = PR[90,1] + 36.831;
   1:  PR[91,2] = PR[90,2] + 26.588;
   1:  PR[91,3] = PR[90,3] + 77.811;
   1:L PR[91] R[100]mm/sec CNT100;
   1:  PR[91,1] = PR[90,1] + 35.284;
   1:  PR[91,2] = PR[90,2] + 26.737;
   1:  PR[91,3] = PR[90,3] + 77.825;
   1:L PR[91] R[100]mm/sec CNT100;
   1:  PR[91,1] = PR[90,1] + 34.661;
   1:  PR[91,2] = PR[90,2] + 26.702;
   1:  PR[91,3] = PR[90,3] + 77.831;
   1:L PR[91] R[100]mm/sec CNT100;
   1:  PR[91,1] = PR[90,1] + 30.172;
   1:  PR[91,2] = PR[90,2] + 26.343;
   1:  PR[91,3] = PR[90,3] + 77.833;
   1:L PR[91] R[100]mm/sec CNT100;
   1:  PR[91,1] = PR[90,1] + 27.461;
   1:  PR[91,2] = PR[90,2] + 25.721;
   1:  PR[91,3] = PR[90,3] + 77.851;
   1:L PR[91] R[100]mm/sec CNT100;
   1:  PR[91,1] = PR[90,1] + 24.763;
   1:  PR[91,2] = PR[90,2] + 25.017;
   1:  PR[91,3] = PR[90,3] + 77.861;
   1:L PR[91] R[100]mm/sec CNT100;
   1:  PR[91,1] = PR[90,1] + 23.172;
   1:  PR[91,2] = PR[90,2] + 25.256;
   1:  PR[91,3] = PR[90,3] + 77.872;
   1:L PR[91] R[100]mm/sec CNT100;
   1:  PR[91,1] = PR[90,1] + 17.573;
   1:  PR[91,2] = PR[90,2] + 25.436;
   1:  PR[91,3] = PR[90,3] + 77.878;
   1:L PR[91] R[100]mm/sec CNT100;
   1:  PR[91,1] = PR[90,1] + 16.833;
   1:  PR[91,2] = PR[90,2] + 25.406;
   1:  PR[91,3] = PR[90,3] + 77.900;
   1:L PR[91] R[100]mm/sec CNT100;
   1:  PR[91,1] = PR[90,1] + 10.865;
   1:  PR[91,2] = PR[90,2] + 24.118;
   1:  PR[91,3] = PR[90,3] + 77.903;
   1:L PR[91] R[100]mm/sec CNT100;
   1:  PR[91,1] = PR[90,1] + 10.534;
   1:  PR[91,2] = PR[90,2] + 24.028;
   1:  PR[91,3] = PR[90,3] + 77.927;
   1:L PR[91] R[100]mm/sec CNT100;
   1:  PR[91,1] = PR[90,1] + 9.578;
   1:  PR[91,2] = PR[90,2] + 23.589;
   1:  PR[91,3] = PR[90,3] + 77.928;
   1:L PR[91] R[100]mm/sec CNT100;
   1:  PR[91,1] = PR[90,1] + 7.992;
   1:  PR[91,2] = PR[90,2] + 23.998;
   1:  PR[91,3] = PR[90,3] + 77.932;
   1:L PR[91] R[100]mm/sec CNT100;
   1:  PR[91,1] = PR[90,1] + 7.478;
   1:  PR[91,2] = PR[90,2] + 24.102;
   1:  PR[91,3] = PR[90,3] + 77.938;
   1:L PR[91] R[100]mm/sec CNT100;
   1:  PR[91,1] = PR[90,1] + 4.632;
   1:  PR[91,2] = PR[90,2] + 24.439;
   1:  PR[91,3] = PR[90,3] + 77.940;
   1:L PR[91] R[100]mm/sec CNT100;
   1:  PR[91,1] = PR[90,1] + 0.604;
   1:  PR[91,2] = PR[90,2] + 24.721;
   1:  PR[91,3] = PR[90,3] + 77.952;
   1:L PR[91] R[100]mm/sec CNT100;
   1:  PR[91,1] = PR[90,1] + -0.800;
   1:  PR[91,2] = PR[90,2] + 24.718;
   1:  PR[91,3] = PR[90,3] + 77.967;
   1:L PR[91] R[100]mm/sec CNT100;
   1:  PR[91,1] = PR[90,1] + -7.222;
   1:  PR[91,2] = PR[90,2] + 24.070;
   1:  PR[91,3] = PR[90,3] + 77.973;
   1:L PR[91] R[100]mm/sec CNT100;
   1:  PR[91,1] = PR[90,1] + -7.972;
   1:  PR[91,2] = PR[90,2] + 23.894;
   1:  PR[91,3] = PR[90,3] + 77.998;
   1:L PR[91] R[100]mm/sec CNT100;
   1:  PR[91,1] = PR[90,1] + -9.821;
   1:  PR[91,2] = PR[90,2] + 24.106;
   1:  PR[91,3] = PR[90,3] + 78.001;
   1:L PR[91] R[100]mm/sec CNT100;
   1:  PR[91,1] = PR[90,1] + -13.981;
   1:  PR[91,2] = PR[90,2] + 24.484;
   1:  PR[91,3] = PR[90,3] + 78.008;
   1:L PR[91] R[100]mm/sec CNT100;
   1:  PR[91,1] = PR[90,1] + -23.990;
   1:  PR[91,2] = PR[90,2] + 24.854;
   1:  PR[91,3] = PR[90,3] + 78.024;
   1:L PR[91] R[100]mm/sec CNT100;
   1:  PR[91,1] = PR[90,1] + -31.838;
   1:  PR[91,2] = PR[90,2] + 24.605;
   1:  PR[91,3] = PR[90,3] + 78.063;
   1:L PR[91] R[100]mm/sec CNT100;
   1:  PR[91,1] = PR[90,1] + -37.491;
   1:  PR[91,2] = PR[90,2] + 24.122;
   1:  PR[91,3] = PR[90,3] + 78.093;
   1:L PR[91] R[100]mm/sec CNT100;
   1:  PR[91,1] = PR[90,1] + -38.823;
   1:  PR[91,2] = PR[90,2] + 23.982;
   1:  PR[91,3] = PR[90,3] + 78.115;
   1:L PR[91] R[100]mm/sec CNT100;
   1:  PR[91,1] = PR[90,1] + -46.088;
   1:  PR[91,2] = PR[90,2] + 22.585;
   1:  PR[91,3] = PR[90,3] + 78.121;
   1:L PR[91] R[100]mm/sec CNT100;
   1:  PR[91,1] = PR[90,1] + -51.135;
   1:  PR[91,2] = PR[90,2] + 21.016;
   1:  PR[91,3] = PR[90,3] + 78.149;
   1:L PR[91] R[100]mm/sec CNT100;
   1:  PR[91,1] = PR[90,1] + -52.570;
   1:  PR[91,2] = PR[90,2] + 20.546;
   1:  PR[91,3] = PR[90,3] + 78.170;
   1:L PR[91] R[100]mm/sec CNT100;
   1:  PR[91,1] = PR[90,1] + -53.318;
   1:  PR[91,2] = PR[90,2] + 20.274;
   1:  PR[91,3] = PR[90,3] + 78.176;
   1:L PR[91] R[100]mm/sec CNT100;
   1:  PR[91,1] = PR[90,1] + -57.031;
   1:  PR[91,2] = PR[90,2] + 18.331;
   1:  PR[91,3] = PR[90,3] + 78.179;
   1:L PR[91] R[100]mm/sec CNT100;
   1:  PR[91] = PR[90];
   1:  PR[91,1] = PR[90,1] + -58.525;
   1:  PR[91,2] = PR[90,2] + 16.939;
   1:  PR[91,3] = PR[90,3] + 79.495;
   1:L PR[91] R[100]mm/sec CNT100;
   1:  PR[91,1] = PR[90,1] + -60.424;
   1:  PR[91,2] = PR[90,2] + 15.436;
   1:  PR[91,3] = PR[90,3] + 78.204;
   1:L PR[91] R[100]mm/sec CNT100;
   1:  PR[91,1] = PR[90,1] + -63.571;
   1:  PR[91,2] = PR[90,2] + 12.823;
   1:  PR[91,3] = PR[90,3] + 78.214;
   1:L PR[91] R[100]mm/sec CNT100;
   1:  PR[91,1] = PR[90,1] + -63.889;
   1:  PR[91,2] = PR[90,2] + 12.432;
   1:  PR[91,3] = PR[90,3] + 78.230;
   1:L PR[91] R[100]mm/sec CNT100;
   1:  PR[91,1] = PR[90,1] + -65.592;
   1:  PR[91,2] = PR[90,2] + 10.265;
   1:  PR[91,3] = PR[90,3] + 78.232;
   1:L PR[91] R[100]mm/sec CNT100;
   1:  PR[91,1] = PR[90,1] + -66.841;
   1:  PR[91,2] = PR[90,2] + 8.515;
   1:  PR[91,3] = PR[90,3] + 78.243;
   1:L PR[91] R[100]mm/sec CNT100;
   1:  PR[91,1] = PR[90,1] + -68.688;
   1:  PR[91,2] = PR[90,2] + 3.945;
   1:  PR[91,3] = PR[90,3] + 78.251;
   1:L PR[91] R[100]mm/sec CNT100;
   1:  PR[91,1] = PR[90,1] + -68.804;
   1:  PR[91,2] = PR[90,2] + 3.058;
   1:  PR[91,3] = PR[90,3] + 78.271;
   1:L PR[91] R[100]mm/sec CNT100;
   1:  PR[91,1] = PR[90,1] + -69.318;
   1:  PR[91,2] = PR[90,2] + 0.144;
   1:  PR[91,3] = PR[90,3] + 78.274;
   1:L PR[91] R[100]mm/sec CNT100;
   1:  PR[91,1] = PR[90,1] + -69.436;
   1:  PR[91,2] = PR[90,2] + -0.725;
   1:  PR[91,3] = PR[90,3] + 78.286;
   1:L PR[91] R[100]mm/sec CNT100;
   1:  PR[91,1] = PR[90,1] + -68.966;
   1:  PR[91,2] = PR[90,2] + -4.088;
   1:  PR[91,3] = PR[90,3] + 78.289;
   1:L PR[91] R[100]mm/sec CNT100;
   1:  PR[91,1] = PR[90,1] + -68.850;
   1:  PR[91,2] = PR[90,2] + -4.728;
   1:  PR[91,3] = PR[90,3] + 78.302;
   1:L PR[91] R[100]mm/sec CNT100;
   1:  PR[91,1] = PR[90,1] + -68.758;
   1:  PR[91,2] = PR[90,2] + -5.058;
   1:  PR[91,3] = PR[90,3] + 78.305;
   1:L PR[91] R[100]mm/sec CNT100;
   1:  PR[91,1] = PR[90,1] + -68.702;
   1:  PR[91,2] = PR[90,2] + -5.478;
   1:  PR[91,3] = PR[90,3] + 78.306;
   1:L PR[91] R[100]mm/sec CNT100;
   1:  PR[91,1] = PR[90,1] + -68.557;
   1:  PR[91,2] = PR[90,2] + -5.829;
   1:  PR[91,3] = PR[90,3] + 78.308;
   1:L PR[91] R[100]mm/sec CNT100;
   1:  PR[91,1] = PR[90,1] + -66.711;
   1:  PR[91,2] = PR[90,2] + -10.010;
   1:  PR[91,3] = PR[90,3] + 78.309;
   1:L PR[91] R[100]mm/sec CNT100;
   1:  PR[91,1] = PR[90,1] + -65.919;
   1:  PR[91,2] = PR[90,2] + -11.101;
   1:  PR[91,3] = PR[90,3] + 78.327;
   1:L PR[91] R[100]mm/sec CNT100;
   1:  PR[91,1] = PR[90,1] + -63.520;
   1:  PR[91,2] = PR[90,2] + -14.179;
   1:  PR[91,3] = PR[90,3] + 78.333;
   1:L PR[91] R[100]mm/sec CNT100;
   1:  PR[91,1] = PR[90,1] + -61.156;
   1:  PR[91,2] = PR[90,2] + -16.312;
   1:  PR[91,3] = PR[90,3] + 78.348;
   1:L PR[91] R[100]mm/sec CNT100;
   1:  PR[91,1] = PR[90,1] + -59.358;
   1:  PR[91,2] = PR[90,2] + -17.811;
   1:  PR[91,3] = PR[90,3] + 78.360;
   1:L PR[91] R[100]mm/sec CNT100;
   1:  PR[91,1] = PR[90,1] + -54.757;
   1:  PR[91,2] = PR[90,2] + -20.631;
   1:  PR[91,3] = PR[90,3] + 78.370;
   1:L PR[91] R[100]mm/sec CNT100;
   1:  PR[91,1] = PR[90,1] + -54.388;
   1:  PR[91,2] = PR[90,2] + -20.832;
   1:  PR[91,3] = PR[90,3] + 78.391;
   1:L PR[91] R[100]mm/sec CNT100;
   1:  PR[91,1] = PR[90,1] + -49.506;
   1:  PR[91,2] = PR[90,2] + -22.657;
   1:  PR[91,3] = PR[90,3] + 78.393;
   1:L PR[91] R[100]mm/sec CNT100;
   1:  PR[91,1] = PR[90,1] + -46.142;
   1:  PR[91,2] = PR[90,2] + -23.805;
   1:  PR[91,3] = PR[90,3] + 78.413;
   1:L PR[91] R[100]mm/sec CNT100;
   1:  PR[91,1] = PR[90,1] + -44.274;
   1:  PR[91,2] = PR[90,2] + -24.235;
   1:  PR[91,3] = PR[90,3] + 78.427;
   1:L PR[91] R[100]mm/sec CNT100;
   1:  PR[91,1] = PR[90,1] + -41.647;
   1:  PR[91,2] = PR[90,2] + -24.752;
   1:  PR[91,3] = PR[90,3] + 78.434;
   1:L PR[91] R[100]mm/sec CNT100;
   1:  PR[91,1] = PR[90,1] + -37.159;
   1:  PR[91,2] = PR[90,2] + -25.586;
   1:  PR[91,3] = PR[90,3] + 78.445;
   1:L PR[91] R[100]mm/sec CNT100;
   1:  PR[91,1] = PR[90,1] + -31.449;
   1:  PR[91,2] = PR[90,2] + -26.196;
   1:  PR[91,3] = PR[90,3] + 78.463;
   1:L PR[91] R[100]mm/sec CNT100;
   1:  PR[91,1] = PR[90,1] + -30.691;
   1:  PR[91,2] = PR[90,2] + -26.257;
   1:  PR[91,3] = PR[90,3] + 78.485;
   1:L PR[91] R[100]mm/sec CNT100;
   1:  PR[91,1] = PR[90,1] + -21.356;
   1:  PR[91,2] = PR[90,2] + -26.566;
   1:  PR[91,3] = PR[90,3] + 78.488;
   1:L PR[91] R[100]mm/sec CNT100;
   1:  PR[91,1] = PR[90,1] + -18.618;
   1:  PR[91,2] = PR[90,2] + -26.480;
   1:  PR[91,3] = PR[90,3] + 78.525;
   1:L PR[91] R[100]mm/sec CNT100;
   1:  PR[91,1] = PR[90,1] + -11.437;
   1:  PR[91,2] = PR[90,2] + -26.211;
   1:  PR[91,3] = PR[90,3] + 78.536;
   1:L PR[91] R[100]mm/sec CNT100;
   1:  PR[91,1] = PR[90,1] + -10.861;
   1:  PR[91,2] = PR[90,2] + -26.169;
   1:  PR[91,3] = PR[90,3] + 78.564;
   1:L PR[91] R[100]mm/sec CNT100;
   1:  PR[91,1] = PR[90,1] + -7.616;
   1:  PR[91,2] = PR[90,2] + -25.801;
   1:  PR[91,3] = PR[90,3] + 78.566;
   1:L PR[91] R[100]mm/sec CNT100;
   1:  PR[91,1] = PR[90,1] + -6.348;
   1:  PR[91,2] = PR[90,2] + -25.766;
   1:  PR[91,3] = PR[90,3] + 78.579;
   1:L PR[91] R[100]mm/sec CNT100;
   1:  PR[91,1] = PR[90,1] + -0.655;
   1:  PR[91,2] = PR[90,2] + -26.360;
   1:  PR[91,3] = PR[90,3] + 78.584;
   1:L PR[91] R[100]mm/sec CNT100;
   1:  PR[91,1] = PR[90,1] + -0.158;
   1:  PR[91,2] = PR[90,2] + -26.392;
   1:  PR[91,3] = PR[90,3] + 78.607;
   1:L PR[91] R[100]mm/sec CNT100;
   1:  PR[91,1] = PR[90,1] + 2.110;
   1:  PR[91,2] = PR[90,2] + -26.397;
   1:  PR[91,3] = PR[90,3] + 78.608;
   1:L PR[91] R[100]mm/sec CNT100;
   1:  PR[91,1] = PR[90,1] + 5.125;
   1:  PR[91,2] = PR[90,2] + -26.188;
   1:  PR[91,3] = PR[90,3] + 78.617;
   1:L PR[91] R[100]mm/sec CNT100;
   1:  PR[91,1] = PR[90,1] + 8.656;
   1:  PR[91,2] = PR[90,2] + -25.770;
   1:  PR[91,3] = PR[90,3] + 78.629;
   1:L PR[91] R[100]mm/sec CNT100;
   1:  PR[91,1] = PR[90,1] + 9.750;
   1:  PR[91,2] = PR[90,2] + -25.548;
   1:  PR[91,3] = PR[90,3] + 78.643;
   1:L PR[91] R[100]mm/sec CNT100;
   1:  PR[91,1] = PR[90,1] + 16.795;
   1:  PR[91,2] = PR[90,2] + -27.065;
   1:  PR[91,3] = PR[90,3] + 78.648;
   1:L PR[91] R[100]mm/sec CNT100;
   1:  PR[91,1] = PR[90,1] + 16.968;
   1:  PR[91,2] = PR[90,2] + -27.072;
   1:  PR[91,3] = PR[90,3] + 78.676;
   1:L PR[91] R[100]mm/sec CNT100;
   1:  PR[91,1] = PR[90,1] + 23.224;
   1:  PR[91,2] = PR[90,2] + -26.871;
   1:  PR[91,3] = PR[90,3] + 78.677;
   1:L PR[91] R[100]mm/sec CNT100;
   1:  PR[91,1] = PR[90,1] + 24.298;
   1:  PR[91,2] = PR[90,2] + -26.713;
   1:  PR[91,3] = PR[90,3] + 78.701;
   1:L PR[91] R[100]mm/sec CNT100;
   1:  PR[91,1] = PR[90,1] + 26.009;
   1:  PR[91,2] = PR[90,2] + -27.159;
   1:  PR[91,3] = PR[90,3] + 78.705;
   1:L PR[91] R[100]mm/sec CNT100;
   1:  PR[91,1] = PR[90,1] + 29.800;
   1:  PR[91,2] = PR[90,2] + -28.028;
   1:  PR[91,3] = PR[90,3] + 78.712;
   1:L PR[91] R[100]mm/sec CNT100;
   1:  PR[91,1] = PR[90,1] + 33.069;
   1:  PR[91,2] = PR[90,2] + -28.289;
   1:  PR[91,3] = PR[90,3] + 78.728;
   1:L PR[91] R[100]mm/sec CNT100;
   1:  PR[91,1] = PR[90,1] + 34.948;
   1:  PR[91,2] = PR[90,2] + -28.395;
   1:  PR[91,3] = PR[90,3] + 78.740;
   1:L PR[91] R[100]mm/sec CNT100;
   1:  PR[91,1] = PR[90,1] + 39.134;
   1:  PR[91,2] = PR[90,2] + -27.994;
   1:  PR[91,3] = PR[90,3] + 78.748;
   1:L PR[91] R[100]mm/sec CNT100;
   1:  PR[91,1] = PR[90,1] + 40.116;
   1:  PR[91,2] = PR[90,2] + -27.918;
   1:  PR[91,3] = PR[90,3] + 78.764;
   1:L PR[91] R[100]mm/sec CNT100;
   1:  PR[91,1] = PR[90,1] + 40.467;
   1:  PR[91,2] = PR[90,2] + -27.858;
   1:  PR[91,3] = PR[90,3] + 78.768;
   1:L PR[91] R[100]mm/sec CNT100;
   1:  PR[91,1] = PR[90,1] + 44.640;
   1:  PR[91,2] = PR[90,2] + -26.858;
   1:  PR[91,3] = PR[90,3] + 78.770;
   1:L PR[91] R[100]mm/sec CNT100;
   1:  PR[91,1] = PR[90,1] + 47.413;
   1:  PR[91,2] = PR[90,2] + -25.928;
   1:  PR[91,3] = PR[90,3] + 78.786;
   1:L PR[91] R[100]mm/sec CNT100;
   1:  PR[91,1] = PR[90,1] + 48.507;
   1:  PR[91,2] = PR[90,2] + -25.470;
   1:  PR[91,3] = PR[90,3] + 78.798;
   1:L PR[91] R[100]mm/sec CNT100;
   1:  PR[91,1] = PR[90,1] + 50.085;
   1:  PR[91,2] = PR[90,2] + -24.647;
   1:  PR[91,3] = PR[90,3] + 78.803;
   1:L PR[91] R[100]mm/sec CNT100;
   1:  PR[91,1] = PR[90,1] + 52.639;
   1:  PR[91,2] = PR[90,2] + -23.567;
   1:  PR[91,3] = PR[90,3] + 78.810;
   1:L PR[91] R[100]mm/sec CNT100;
   1:  PR[91,1] = PR[90,1] + 54.654;
   1:  PR[91,2] = PR[90,2] + -22.457;
   1:  PR[91,3] = PR[90,3] + 78.820;
   1:L PR[91] R[100]mm/sec CNT100;
   1:  PR[91,1] = PR[90,1] + 56.192;
   1:  PR[91,2] = PR[90,2] + -21.524;
   1:  PR[91,3] = PR[90,3] + 78.829;
   1:L PR[91] R[100]mm/sec CNT100;
   1:  PR[91,1] = PR[90,1] + 57.560;
   1:  PR[91,2] = PR[90,2] + -20.498;
   1:  PR[91,3] = PR[90,3] + 78.837;
   1:L PR[91] R[100]mm/sec CNT100;
   1:  PR[91,1] = PR[90,1] + 59.786;
   1:  PR[91,2] = PR[90,2] + -19.072;
   1:  PR[91,3] = PR[90,3] + 78.843;
   1:L PR[91] R[100]mm/sec CNT100;
   1:  PR[91,1] = PR[90,1] + 62.571;
   1:  PR[91,2] = PR[90,2] + -16.719;
   1:  PR[91,3] = PR[90,3] + 78.854;
   1:L PR[91] R[100]mm/sec CNT100;
   1:  PR[91,1] = PR[90,1] + 63.263;
   1:  PR[91,2] = PR[90,2] + -16.116;
   1:  PR[91,3] = PR[90,3] + 78.868;
   1:L PR[91] R[100]mm/sec CNT100;
   1:  PR[91,1] = PR[90,1] + 63.827;
   1:  PR[91,2] = PR[90,2] + -15.457;
   1:  PR[91,3] = PR[90,3] + 78.872;
   1:L PR[91] R[100]mm/sec CNT100;
   1:  PR[91,1] = PR[90,1] + 66.315;
   1:  PR[91,2] = PR[90,2] + -12.369;
   1:  PR[91,3] = PR[90,3] + 78.875;
   1:L PR[91] R[100]mm/sec CNT100;
   1:  PR[91,1] = PR[90,1] + 67.947;
   1:  PR[91,2] = PR[90,2] + -9.434;
   1:  PR[91,3] = PR[90,3] + 78.890;
   1:L PR[91] R[100]mm/sec CNT100;
   1:  PR[91,1] = PR[90,1] + 68.606;
   1:  PR[91,2] = PR[90,2] + -7.928;
   1:  PR[91,3] = PR[90,3] + 78.904;
   1:L PR[91] R[100]mm/sec CNT100;
   1:  PR[91,1] = PR[90,1] + 69.456;
   1:  PR[91,2] = PR[90,2] + -5.289;
   1:  PR[91,3] = PR[90,3] + 78.910;
   1:L PR[91] R[100]mm/sec CNT100;
   1:  PR[91,1] = PR[90,1] + 69.757;
   1:  PR[91,2] = PR[90,2] + -3.183;
   1:  PR[91,3] = PR[90,3] + 78.921;
   1:L PR[91] R[100]mm/sec CNT100;
   1:  PR[91,1] = PR[90,1] + 70.012;
   1:  PR[91,2] = PR[90,2] + -0.768;
   1:  PR[91,3] = PR[90,3] + 78.929;
   1:L PR[91] R[100]mm/sec CNT100;
   1:  PR[91,1] = PR[90,1] + 69.706;
   1:  PR[91,2] = PR[90,2] + 1.349;
   1:  PR[91,3] = PR[90,3] + 78.939;
   1:L PR[91] R[100]mm/sec CNT100;
   1:  PR[91,1] = PR[90,1] + 69.445;
   1:  PR[91,2] = PR[90,2] + 3.866;
   1:  PR[91,3] = PR[90,3] + 78.947;
   1:L PR[91] R[100]mm/sec CNT100;
   1:  PR[91,1] = PR[90,1] + 68.606;
   1:  PR[91,2] = PR[90,2] + 6.468;
   1:  PR[91,3] = PR[90,3] + 78.957;
   1:L PR[91] R[100]mm/sec CNT100;
   1:  PR[91,1] = PR[90,1] + 67.947;
   1:  PR[91,2] = PR[90,2] + 7.974;
   1:  PR[91,3] = PR[90,3] + 78.968;
   1:L PR[91] R[100]mm/sec CNT100;
   1:  PR[91,1] = PR[90,1] + 66.308;
   1:  PR[91,2] = PR[90,2] + 10.922;
   1:  PR[91,3] = PR[90,3] + 78.974;
   1:L PR[91] R[100]mm/sec CNT100;
   1:  PR[91,1] = PR[90,1] + 65.847;
   1:  PR[91,2] = PR[90,2] + 11.513;
   1:  PR[91,3] = PR[90,3] + 78.988;
   1:L PR[91] R[100]mm/sec CNT100;
   1:  PR[91,1] = PR[90,1] + 63.829;
   1:  PR[91,2] = PR[90,2] + 13.995;
   1:  PR[91,3] = PR[90,3] + 78.991;
   1:L PR[91] R[100]mm/sec CNT100;
   1:  PR[91,1] = PR[90,1] + 63.263;
   1:  PR[91,2] = PR[90,2] + 14.657;
   1:  PR[91,3] = PR[90,3] + 79.003;
   1:L PR[91] R[100]mm/sec CNT100;
   1:  PR[91,1] = PR[90,1] + 62.571;
   1:  PR[91,2] = PR[90,2] + 15.260;
   1:  PR[91,3] = PR[90,3] + 79.007;
   1:L PR[91] R[100]mm/sec CNT100;
   1:  PR[91,1] = PR[90,1] + 59.786;
   1:  PR[91,2] = PR[90,2] + 17.613;
   1:  PR[91,3] = PR[90,3] + 79.010;
   1:L PR[91] R[100]mm/sec CNT100;
   1:  PR[91,1] = PR[90,1] + 57.560;
   1:  PR[91,2] = PR[90,2] + 19.039;
   1:  PR[91,3] = PR[90,3] + 79.024;
   1:L PR[91] R[100]mm/sec CNT100;
   1:  PR[91,1] = PR[90,1] + 56.192;
   1:  PR[91,2] = PR[90,2] + 20.065;
   1:  PR[91,3] = PR[90,3] + 79.035;
   1:L PR[91] R[100]mm/sec CNT100;
   1:  PR[91,1] = PR[90,1] + 54.654;
   1:  PR[91,2] = PR[90,2] + 20.998;
   1:  PR[91,3] = PR[90,3] + 79.042;
   1:L PR[91] R[100]mm/sec CNT100;
   1:  PR[91,1] = PR[90,1] + 52.639;
   1:  PR[91,2] = PR[90,2] + 22.108;
   1:  PR[91,3] = PR[90,3] + 79.049;
   1:L PR[91] R[100]mm/sec CNT100;
   1:  PR[91,1] = PR[90,1] + 50.085;
   1:  PR[91,2] = PR[90,2] + 23.189;
   1:  PR[91,3] = PR[90,3] + 79.058;
   1:L PR[91] R[100]mm/sec CNT100;
   1:  PR[91,1] = PR[90,1] + 48.507;
   1:  PR[91,2] = PR[90,2] + 24.012;
   1:  PR[91,3] = PR[90,3] + 79.069;
   1:L PR[91] R[100]mm/sec CNT100;
   1:  PR[91,1] = PR[90,1] + 47.413;
   1:  PR[91,2] = PR[90,2] + 24.469;
   1:  PR[91,3] = PR[90,3] + 79.075;
   1:L PR[91] R[100]mm/sec CNT100;
   1:  PR[91,1] = PR[90,1] + 44.640;
   1:  PR[91,2] = PR[90,2] + 25.399;
   1:  PR[91,3] = PR[90,3] + 79.080;
   1:L PR[91] R[100]mm/sec CNT100;
   1:  PR[91,1] = PR[90,1] + 40.467;
   1:  PR[91,2] = PR[90,2] + 26.399;
   1:  PR[91,3] = PR[90,3] + 79.092;
   1:L PR[91] R[100]mm/sec CNT100;
   1:  PR[91,1] = PR[90,1] + 40.116;
   1:  PR[91,2] = PR[90,2] + 26.460;
   1:  PR[91,3] = PR[90,3] + 79.108;
   1:L PR[91] R[100]mm/sec CNT100;
   1:  PR[91,1] = PR[90,1] + 39.134;
   1:  PR[91,2] = PR[90,2] + 26.535;
   1:  PR[91,3] = PR[90,3] + 79.110;
   1:L PR[91] R[100]mm/sec CNT100;
   1:  PR[91,1] = PR[90,1] + 34.948;
   1:  PR[91,2] = PR[90,2] + 26.936;
   1:  PR[91,3] = PR[90,3] + 79.114;
   1:L PR[91] R[100]mm/sec CNT100;
   1:  PR[91,1] = PR[90,1] + 33.069;
   1:  PR[91,2] = PR[90,2] + 26.830;
   1:  PR[91,3] = PR[90,3] + 79.130;
   1:L PR[91] R[100]mm/sec CNT100;
   1:  PR[91,1] = PR[90,1] + 29.800;
   1:  PR[91,2] = PR[90,2] + 26.569;
   1:  PR[91,3] = PR[90,3] + 79.138;
   1:L PR[91] R[100]mm/sec CNT100;
   1:  PR[91,1] = PR[90,1] + 26.009;
   1:  PR[91,2] = PR[90,2] + 25.701;
   1:  PR[91,3] = PR[90,3] + 79.150;
   1:L PR[91] R[100]mm/sec CNT100;
   1:  PR[91,1] = PR[90,1] + 24.298;
   1:  PR[91,2] = PR[90,2] + 25.254;
   1:  PR[91,3] = PR[90,3] + 79.166;
   1:L PR[91] R[100]mm/sec CNT100;
   1:  PR[91,1] = PR[90,1] + 23.224;
   1:  PR[91,2] = PR[90,2] + 25.412;
   1:  PR[91,3] = PR[90,3] + 79.173;
   1:L PR[91] R[100]mm/sec CNT100;
   1:  PR[91,1] = PR[90,1] + 16.968;
   1:  PR[91,2] = PR[90,2] + 25.613;
   1:  PR[91,3] = PR[90,3] + 79.177;
   1:L PR[91] R[100]mm/sec CNT100;
   1:  PR[91,1] = PR[90,1] + 16.795;
   1:  PR[91,2] = PR[90,2] + 25.606;
   1:  PR[91,3] = PR[90,3] + 79.202;
   1:L PR[91] R[100]mm/sec CNT100;
   1:  PR[91,1] = PR[90,1] + 9.750;
   1:  PR[91,2] = PR[90,2] + 24.089;
   1:L PR[91] R[100]mm/sec CNT100;
   1:  PR[91,1] = PR[90,1] + 8.665;
   1:  PR[91,2] = PR[90,2] + 24.309;
   1:  PR[91,3] = PR[90,3] + 79.230;
   1:L PR[91] R[100]mm/sec CNT100;
   1:  PR[91,1] = PR[90,1] + 5.140;
   1:  PR[91,2] = PR[90,2] + 24.727;
   1:  PR[91,3] = PR[90,3] + 79.235;
   1:L PR[91] R[100]mm/sec CNT100;
   1:  PR[91,1] = PR[90,1] + 2.127;
   1:  PR[91,2] = PR[90,2] + 24.938;
   1:  PR[91,3] = PR[90,3] + 79.249;
   1:L PR[91] R[100]mm/sec CNT100;
   1:  PR[91,1] = PR[90,1] + -0.101;
   1:  PR[91,2] = PR[90,2] + 24.933;
   1:  PR[91,3] = PR[90,3] + 79.261;
   1:L PR[91] R[100]mm/sec CNT100;
   1:  PR[91,1] = PR[90,1] + -6.393;
   1:  PR[91,2] = PR[90,2] + 24.297;
   1:  PR[91,3] = PR[90,3] + 79.269;
   1:L PR[91] R[100]mm/sec CNT100;
   1:  PR[91,1] = PR[90,1] + -11.231;
   1:  PR[91,2] = PR[90,2] + 24.737;
   1:  PR[91,3] = PR[90,3] + 79.294;
   1:L PR[91] R[100]mm/sec CNT100;
   1:  PR[91,1] = PR[90,1] + -18.619;
   1:  PR[91,2] = PR[90,2] + 25.021;
   1:  PR[91,3] = PR[90,3] + 79.313;
   1:L PR[91] R[100]mm/sec CNT100;
   1:  PR[91,1] = PR[90,1] + -21.356;
   1:  PR[91,2] = PR[90,2] + 25.107;
   1:  PR[91,3] = PR[90,3] + 79.342;
   1:L PR[91] R[100]mm/sec CNT100;
   1:  PR[91,1] = PR[90,1] + -30.684;
   1:  PR[91,2] = PR[90,2] + 24.799;
   1:  PR[91,3] = PR[90,3] + 79.353;
   1:L PR[91] R[100]mm/sec CNT100;
   1:  PR[91,1] = PR[90,1] + -31.732;
   1:  PR[91,2] = PR[90,2] + 24.710;
   1:  PR[91,3] = PR[90,3] + 79.390;
   1:L PR[91] R[100]mm/sec CNT100;
   1:  PR[91,1] = PR[90,1] + -37.259;
   1:  PR[91,2] = PR[90,2] + 24.127;
   1:  PR[91,3] = PR[90,3] + 79.394;
   1:L PR[91] R[100]mm/sec CNT100;
   1:  PR[91,1] = PR[90,1] + -44.886;
   1:  PR[91,2] = PR[90,2] + 22.670;
   1:  PR[91,3] = PR[90,3] + 79.416;
   1:L PR[91] R[100]mm/sec CNT100;
   1:  PR[91,1] = PR[90,1] + -51.856;
   1:  PR[91,2] = PR[90,2] + 20.497;
   1:  PR[91,3] = PR[90,3] + 79.446;
   1:L PR[91] R[100]mm/sec CNT100;
   1:  PR[91,1] = PR[90,1] + -56.441;
   1:  PR[91,2] = PR[90,2] + 18.105;
   1:  PR[91,3] = PR[90,3] + 79.475;
   1:L PR[91] R[100]mm/sec CNT100;
   1:  PR[91] = PR[90];
   1:  PR[91,1] = PR[90,1] + -57.127;
   1:  PR[91,2] = PR[90,2] + 17.164;
   1:  PR[91,3] = PR[90,3] + 80.795;
   1:L PR[91] R[100]mm/sec CNT100;
   1:  PR[91,1] = PR[90,1] + -59.761;
   1:  PR[91,2] = PR[90,2] + 15.080;
   1:  PR[91,3] = PR[90,3] + 79.501;
   1:L PR[91] R[100]mm/sec CNT100;
   1:  PR[91,1] = PR[90,1] + -62.266;
   1:  PR[91,2] = PR[90,2] + 13.000;
   1:  PR[91,3] = PR[90,3] + 79.514;
   1:L PR[91] R[100]mm/sec CNT100;
   1:  PR[91,1] = PR[90,1] + -63.125;
   1:  PR[91,2] = PR[90,2] + 11.946;
   1:  PR[91,3] = PR[90,3] + 79.527;
   1:L PR[91] R[100]mm/sec CNT100;
   1:  PR[91,1] = PR[90,1] + -65.801;
   1:  PR[91,2] = PR[90,2] + 8.538;
   1:  PR[91,3] = PR[90,3] + 79.532;
   1:L PR[91] R[100]mm/sec CNT100;
   1:  PR[91,1] = PR[90,1] + -66.670;
   1:  PR[91,2] = PR[90,2] + 6.598;
   1:  PR[91,3] = PR[90,3] + 79.550;
   1:L PR[91] R[100]mm/sec CNT100;
   1:  PR[91,1] = PR[90,1] + -67.726;
   1:  PR[91,2] = PR[90,2] + 3.985;
   1:  PR[91,3] = PR[90,3] + 79.558;
   1:L PR[91] R[100]mm/sec CNT100;
   1:  PR[91,1] = PR[90,1] + -67.747;
   1:  PR[91,2] = PR[90,2] + 3.823;
   1:  PR[91,3] = PR[90,3] + 79.569;
   1:L PR[91] R[100]mm/sec CNT100;
   1:  PR[91,1] = PR[90,1] + -67.921;
   1:  PR[91,2] = PR[90,2] + 2.835;
   1:  PR[91,3] = PR[90,3] + 79.570;
   1:L PR[91] R[100]mm/sec CNT100;
   1:  PR[91,1] = PR[90,1] + -68.404;
   1:  PR[91,2] = PR[90,2] + -0.725;
   1:  PR[91,3] = PR[90,3] + 79.574;
   1:L PR[91] R[100]mm/sec CNT100;
   1:  PR[91,1] = PR[90,1] + -68.209;
   1:  PR[91,2] = PR[90,2] + -2.121;
   1:  PR[91,3] = PR[90,3] + 79.588;
   1:L PR[91] R[100]mm/sec CNT100;
   1:  PR[91,1] = PR[90,1] + -67.922;
   1:  PR[91,2] = PR[90,2] + -3.706;
   1:  PR[91,3] = PR[90,3] + 79.594;
   1:L PR[91] R[100]mm/sec CNT100;
   1:  PR[91,1] = PR[90,1] + -67.733;
   1:  PR[91,2] = PR[90,2] + -4.386;
   1:  PR[91,3] = PR[90,3] + 79.600;
   1:L PR[91] R[100]mm/sec CNT100;
   1:  PR[91,1] = PR[90,1] + -67.589;
   1:  PR[91,2] = PR[90,2] + -5.467;
   1:  PR[91,3] = PR[90,3] + 79.603;
   1:L PR[91] R[100]mm/sec CNT100;
   1:  PR[91,1] = PR[90,1] + -67.132;
   1:  PR[91,2] = PR[90,2] + -6.573;
   1:  PR[91,3] = PR[90,3] + 79.607;
   1:L PR[91] R[100]mm/sec CNT100;
   1:  PR[91,1] = PR[90,1] + -65.623;
   1:  PR[91,2] = PR[90,2] + -9.993;
   1:  PR[91,3] = PR[90,3] + 79.612;
   1:L PR[91] R[100]mm/sec CNT100;
   1:  PR[91,1] = PR[90,1] + -64.279;
   1:  PR[91,2] = PR[90,2] + -11.843;
   1:  PR[91,3] = PR[90,3] + 79.627;
   1:L PR[91] R[100]mm/sec CNT100;
   1:  PR[91,1] = PR[90,1] + -62.471;
   1:  PR[91,2] = PR[90,2] + -14.163;
   1:  PR[91,3] = PR[90,3] + 79.636;
   1:L PR[91] R[100]mm/sec CNT100;
   1:  PR[91,1] = PR[90,1] + -59.300;
   1:  PR[91,2] = PR[90,2] + -17.023;
   1:  PR[91,3] = PR[90,3] + 79.648;
   1:L PR[91] R[100]mm/sec CNT100;
   1:  PR[91,1] = PR[90,1] + -58.360;
   1:  PR[91,2] = PR[90,2] + -17.807;
   1:  PR[91,3] = PR[90,3] + 79.665;
   1:L PR[91] R[100]mm/sec CNT100;
   1:  PR[91,1] = PR[90,1] + -55.860;
   1:  PR[91,2] = PR[90,2] + -19.339;
   1:  PR[91,3] = PR[90,3] + 79.670;
   1:L PR[91] R[100]mm/sec CNT100;
   1:  PR[91,1] = PR[90,1] + -53.634;
   1:  PR[91,2] = PR[90,2] + -20.570;
   1:  PR[91,3] = PR[90,3] + 79.681;
   1:L PR[91] R[100]mm/sec CNT100;
   1:  PR[91,1] = PR[90,1] + -52.629;
   1:  PR[91,2] = PR[90,2] + -21.092;
   1:  PR[91,3] = PR[90,3] + 79.691;
   1:L PR[91] R[100]mm/sec CNT100;
   1:  PR[91,1] = PR[90,1] + -48.737;
   1:  PR[91,2] = PR[90,2] + -22.548;
   1:  PR[91,3] = PR[90,3] + 79.696;
   1:L PR[91] R[100]mm/sec CNT100;
   1:  PR[91,1] = PR[90,1] + -44.199;
   1:  PR[91,2] = PR[90,2] + -24.096;
   1:  PR[91,3] = PR[90,3] + 79.712;
   1:L PR[91] R[100]mm/sec CNT100;
   1:  PR[91,1] = PR[90,1] + -43.532;
   1:  PR[91,2] = PR[90,2] + -24.250;
   1:  PR[91,3] = PR[90,3] + 79.731;
   1:L PR[91] R[100]mm/sec CNT100;
   1:  PR[91,1] = PR[90,1] + -42.508;
   1:  PR[91,2] = PR[90,2] + -24.451;
   1:  PR[91,3] = PR[90,3] + 79.734;
   1:L PR[91] R[100]mm/sec CNT100;
   1:  PR[91,1] = PR[90,1] + -35.626;
   1:  PR[91,2] = PR[90,2] + -25.731;
   1:  PR[91,3] = PR[90,3] + 79.738;
   1:L PR[91] R[100]mm/sec CNT100;
   1:  PR[91,1] = PR[90,1] + -28.455;
   1:  PR[91,2] = PR[90,2] + -26.491;
   1:  PR[91,3] = PR[90,3] + 79.766;
   1:L PR[91] R[100]mm/sec CNT100;
   1:  PR[91,1] = PR[90,1] + -18.729;
   1:  PR[91,2] = PR[90,2] + -26.818;
   1:  PR[91,3] = PR[90,3] + 79.795;
   1:L PR[91] R[100]mm/sec CNT100;
   1:  PR[91,1] = PR[90,1] + -14.970;
   1:  PR[91,2] = PR[90,2] + -26.700;
   1:  PR[91,3] = PR[90,3] + 79.833;
   1:L PR[91] R[100]mm/sec CNT100;
   1:  PR[91,1] = PR[90,1] + -8.725;
   1:  PR[91,2] = PR[90,2] + -26.466;
   1:  PR[91,3] = PR[90,3] + 79.848;
   1:L PR[91] R[100]mm/sec CNT100;
   1:  PR[91,1] = PR[90,1] + -8.035;
   1:  PR[91,2] = PR[90,2] + -26.416;
   1:  PR[91,3] = PR[90,3] + 79.873;
   1:L PR[91] R[100]mm/sec CNT100;
   1:  PR[91,1] = PR[90,1] + -5.547;
   1:  PR[91,2] = PR[90,2] + -26.134;
   1:  PR[91,3] = PR[90,3] + 79.876;
   1:L PR[91] R[100]mm/sec CNT100;
   1:  PR[91,1] = PR[90,1] + -4.527;
   1:  PR[91,2] = PR[90,2] + -26.106;
   1:  PR[91,3] = PR[90,3] + 79.886;
   1:L PR[91] R[100]mm/sec CNT100;
   1:  PR[91,1] = PR[90,1] + -0.160;
   1:  PR[91,2] = PR[90,2] + -26.561;
   1:  PR[91,3] = PR[90,3] + 79.890;
   1:L PR[91] R[100]mm/sec CNT100;
   1:  PR[91,1] = PR[90,1] + 0.543;
   1:  PR[91,2] = PR[90,2] + -26.607;
   1:  PR[91,3] = PR[90,3] + 79.907;
   1:L PR[91] R[100]mm/sec CNT100;
   1:  PR[91,1] = PR[90,1] + 3.638;
   1:  PR[91,2] = PR[90,2] + -26.613;
   1:  PR[91,3] = PR[90,3] + 79.910;
   1:L PR[91] R[100]mm/sec CNT100;
   1:  PR[91,1] = PR[90,1] + 5.637;
   1:  PR[91,2] = PR[90,2] + -26.475;
   1:  PR[91,3] = PR[90,3] + 79.922;
   1:L PR[91] R[100]mm/sec CNT100;
   1:  PR[91,1] = PR[90,1] + 10.246;
   1:  PR[91,2] = PR[90,2] + -25.930;
   1:  PR[91,3] = PR[90,3] + 79.930;
   1:L PR[91] R[100]mm/sec CNT100;
   1:  PR[91,1] = PR[90,1] + 16.533;
   1:  PR[91,2] = PR[90,2] + -27.222;
   1:  PR[91,3] = PR[90,3] + 79.949;
   1:L PR[91] R[100]mm/sec CNT100;
   1:  PR[91,1] = PR[90,1] + 16.683;
   1:  PR[91,2] = PR[90,2] + -27.244;
   1:  PR[91,3] = PR[90,3] + 79.974;
   1:L PR[91] R[100]mm/sec CNT100;
   1:  PR[91,1] = PR[90,1] + 23.285;
   1:  PR[91,2] = PR[90,2] + -27.027;
   1:  PR[91,3] = PR[90,3] + 79.975;
   1:L PR[91] R[100]mm/sec CNT100;
   1:  PR[91,1] = PR[90,1] + 23.841;
   1:  PR[91,2] = PR[90,2] + -26.952;
   1:  PR[91,3] = PR[90,3] + 80.001;
   1:L PR[91] R[100]mm/sec CNT100;
   1:  PR[91,1] = PR[90,1] + 24.558;
   1:  PR[91,2] = PR[90,2] + -27.139;
   1:  PR[91,3] = PR[90,3] + 80.003;
   1:L PR[91] R[100]mm/sec CNT100;
   1:  PR[91,1] = PR[90,1] + 29.428;
   1:  PR[91,2] = PR[90,2] + -28.254;
   1:  PR[91,3] = PR[90,3] + 80.006;
   1:L PR[91] R[100]mm/sec CNT100;
   1:  PR[91,1] = PR[90,1] + 31.477;
   1:  PR[91,2] = PR[90,2] + -28.418;
   1:  PR[91,3] = PR[90,3] + 80.026;
   1:L PR[91] R[100]mm/sec CNT100;
   1:  PR[91,1] = PR[90,1] + 34.612;
   1:  PR[91,2] = PR[90,2] + -28.595;
   1:  PR[91,3] = PR[90,3] + 80.034;
   1:L PR[91] R[100]mm/sec CNT100;
   1:  PR[91,1] = PR[90,1] + 39.040;
   1:  PR[91,2] = PR[90,2] + -28.171;
   1:  PR[91,3] = PR[90,3] + 80.047;
   1:L PR[91] R[100]mm/sec CNT100;
   1:  PR[91,1] = PR[90,1] + 39.704;
   1:  PR[91,2] = PR[90,2] + -28.096;
   1:  PR[91,3] = PR[90,3] + 80.064;
   1:L PR[91] R[100]mm/sec CNT100;
   1:  PR[91,1] = PR[90,1] + 41.112;
   1:  PR[91,2] = PR[90,2] + -27.706;
   1:  PR[91,3] = PR[90,3] + 80.067;
   1:L PR[91] R[100]mm/sec CNT100;
   1:  PR[91,1] = PR[90,1] + 44.509;
   1:  PR[91,2] = PR[90,2] + -26.892;
   1:  PR[91,3] = PR[90,3] + 80.073;
   1:L PR[91] R[100]mm/sec CNT100;
   1:  PR[91,1] = PR[90,1] + 46.070;
   1:  PR[91,2] = PR[90,2] + -26.368;
   1:  PR[91,3] = PR[90,3] + 80.087;
   1:L PR[91] R[100]mm/sec CNT100;
   1:  PR[91,1] = PR[90,1] + 48.476;
   1:  PR[91,2] = PR[90,2] + -25.364;
   1:  PR[91,3] = PR[90,3] + 80.093;
   1:L PR[91] R[100]mm/sec CNT100;
   1:  PR[91,1] = PR[90,1] + 51.725;
   1:  PR[91,2] = PR[90,2] + -23.668;
   1:  PR[91,3] = PR[90,3] + 80.104;
   1:L PR[91] R[100]mm/sec CNT100;
   1:  PR[91,1] = PR[90,1] + 52.139;
   1:  PR[91,2] = PR[90,2] + -23.493;
   1:  PR[91,3] = PR[90,3] + 80.118;
   1:L PR[91] R[100]mm/sec CNT100;
   1:  PR[91,1] = PR[90,1] + 52.374;
   1:  PR[91,2] = PR[90,2] + -23.364;
   1:  PR[91,3] = PR[90,3] + 80.120;
   1:L PR[91] R[100]mm/sec CNT100;
   1:  PR[91,1] = PR[90,1] + 55.803;
   1:  PR[91,2] = PR[90,2] + -21.284;
   1:  PR[91,3] = PR[90,3] + 80.121;
   1:L PR[91] R[100]mm/sec CNT100;
   1:  PR[91,1] = PR[90,1] + 58.756;
   1:  PR[91,2] = PR[90,2] + -19.070;
   1:  PR[91,3] = PR[90,3] + 80.137;
   1:L PR[91] R[100]mm/sec CNT100;
   1:  PR[91,1] = PR[90,1] + 58.864;
   1:  PR[91,2] = PR[90,2] + -19.001;
   1:  PR[91,3] = PR[90,3] + 80.152;
   1:L PR[91] R[100]mm/sec CNT100;
   1:  PR[91,1] = PR[90,1] + 62.286;
   1:  PR[91,2] = PR[90,2] + -16.027;
   1:L PR[91] R[100]mm/sec CNT100;
   1:  PR[91,1] = PR[90,1] + 65.022;
   1:  PR[91,2] = PR[90,2] + -12.827;
   1:  PR[91,3] = PR[90,3] + 80.170;
   1:L PR[91] R[100]mm/sec CNT100;
   1:  PR[91,1] = PR[90,1] + 65.182;
   1:  PR[91,2] = PR[90,2] + -12.628;
   1:  PR[91,3] = PR[90,3] + 80.187;
   1:L PR[91] R[100]mm/sec CNT100;
   1:  PR[91,1] = PR[90,1] + 67.131;
   1:  PR[91,2] = PR[90,2] + -9.121;
   1:  PR[91,3] = PR[90,3] + 80.188;
   1:L PR[91] R[100]mm/sec CNT100;
   1:  PR[91,1] = PR[90,1] + 67.452;
   1:  PR[91,2] = PR[90,2] + -8.389;
   1:  PR[91,3] = PR[90,3] + 80.204;
   1:L PR[91] R[100]mm/sec CNT100;
   1:  PR[91,1] = PR[90,1] + 68.507;
   1:  PR[91,2] = PR[90,2] + -5.114;
   1:  PR[91,3] = PR[90,3] + 80.207;
   1:L PR[91] R[100]mm/sec CNT100;
   1:  PR[91,1] = PR[90,1] + 68.691;
   1:  PR[91,2] = PR[90,2] + -3.827;
   1:  PR[91,3] = PR[90,3] + 80.221;
   1:L PR[91] R[100]mm/sec CNT100;
   1:  PR[91,1] = PR[90,1] + 69.013;
   1:  PR[91,2] = PR[90,2] + -0.768;
   1:  PR[91,3] = PR[90,3] + 80.226;
   1:L PR[91] R[100]mm/sec CNT100;
   1:  PR[91,1] = PR[90,1] + 68.818;
   1:  PR[91,2] = PR[90,2] + 0.583;
   1:  PR[91,3] = PR[90,3] + 80.238;
   1:L PR[91] R[100]mm/sec CNT100;
   1:  PR[91,1] = PR[90,1] + 68.495;
   1:  PR[91,2] = PR[90,2] + 3.691;
   1:  PR[91,3] = PR[90,3] + 80.243;
   1:L PR[91] R[100]mm/sec CNT100;
   1:  PR[91,1] = PR[90,1] + 67.452;
   1:  PR[91,2] = PR[90,2] + 6.930;
   1:  PR[91,3] = PR[90,3] + 80.256;
   1:L PR[91] R[100]mm/sec CNT100;
   1:  PR[91,1] = PR[90,1] + 67.132;
   1:  PR[91,2] = PR[90,2] + 7.661;
   1:  PR[91,3] = PR[90,3] + 80.269;
   1:L PR[91] R[100]mm/sec CNT100;
   1:  PR[91,1] = PR[90,1] + 65.182;
   1:  PR[91,2] = PR[90,2] + 11.169;
   1:  PR[91,3] = PR[90,3] + 80.272;
   1:L PR[91] R[100]mm/sec CNT100;
   1:  PR[91,1] = PR[90,1] + 65.022;
   1:  PR[91,2] = PR[90,2] + 11.368;
   1:  PR[91,3] = PR[90,3] + 80.288;
   1:L PR[91] R[100]mm/sec CNT100;
   1:  PR[91,1] = PR[90,1] + 62.286;
   1:  PR[91,2] = PR[90,2] + 14.568;
   1:  PR[91,3] = PR[90,3] + 80.289;
   1:L PR[91] R[100]mm/sec CNT100;
   1:  PR[91,1] = PR[90,1] + 58.864;
   1:  PR[91,2] = PR[90,2] + 17.542;
   1:  PR[91,3] = PR[90,3] + 80.306;
   1:L PR[91] R[100]mm/sec CNT100;
   1:  PR[91,1] = PR[90,1] + 58.756;
   1:  PR[91,2] = PR[90,2] + 17.612;
   1:  PR[91,3] = PR[90,3] + 80.324;
   1:L PR[91] R[100]mm/sec CNT100;
   1:  PR[91,1] = PR[90,1] + 55.803;
   1:  PR[91,2] = PR[90,2] + 19.826;
   1:  PR[91,3] = PR[90,3] + 80.325;
   1:L PR[91] R[100]mm/sec CNT100;
   1:  PR[91,1] = PR[90,1] + 52.374;
   1:  PR[91,2] = PR[90,2] + 21.905;
   1:  PR[91,3] = PR[90,3] + 80.339;
   1:L PR[91] R[100]mm/sec CNT100;
   1:  PR[91,1] = PR[90,1] + 52.139;
   1:  PR[91,2] = PR[90,2] + 22.034;
   1:  PR[91,3] = PR[90,3] + 80.355;
   1:L PR[91] R[100]mm/sec CNT100;
   1:  PR[91,1] = PR[90,1] + 51.725;
   1:  PR[91,2] = PR[90,2] + 22.209;
   1:  PR[91,3] = PR[90,3] + 80.356;
   1:L PR[91] R[100]mm/sec CNT100;
   1:  PR[91,1] = PR[90,1] + 48.476;
   1:  PR[91,2] = PR[90,2] + 23.905;
   1:  PR[91,3] = PR[90,3] + 80.358;
   1:L PR[91] R[100]mm/sec CNT100;
   1:  PR[91,1] = PR[90,1] + 46.070;
   1:  PR[91,2] = PR[90,2] + 24.909;
   1:  PR[91,3] = PR[90,3] + 80.373;
   1:L PR[91] R[100]mm/sec CNT100;
   1:  PR[91,1] = PR[90,1] + 44.509;
   1:  PR[91,2] = PR[90,2] + 25.434;
   1:  PR[91,3] = PR[90,3] + 80.383;
   1:L PR[91] R[100]mm/sec CNT100;
   1:  PR[91,1] = PR[90,1] + 41.112;
   1:  PR[91,2] = PR[90,2] + 26.248;
   1:  PR[91,3] = PR[90,3] + 80.390;
   1:L PR[91] R[100]mm/sec CNT100;
   1:  PR[91,1] = PR[90,1] + 39.704;
   1:  PR[91,2] = PR[90,2] + 26.637;
   1:  PR[91,3] = PR[90,3] + 80.403;
   1:L PR[91] R[100]mm/sec CNT100;
   1:  PR[91,1] = PR[90,1] + 39.040;
   1:  PR[91,2] = PR[90,2] + 26.712;
   1:  PR[91,3] = PR[90,3] + 80.409;
   1:L PR[91] R[100]mm/sec CNT100;
   1:  PR[91,1] = PR[90,1] + 34.612;
   1:  PR[91,2] = PR[90,2] + 27.136;
   1:  PR[91,3] = PR[90,3] + 80.412;
   1:L PR[91] R[100]mm/sec CNT100;
   1:  PR[91,1] = PR[90,1] + 31.477;
   1:  PR[91,2] = PR[90,2] + 26.959;
   1:  PR[91,3] = PR[90,3] + 80.430;
   1:L PR[91] R[100]mm/sec CNT100;
   1:  PR[91,1] = PR[90,1] + 29.428;
   1:  PR[91,2] = PR[90,2] + 26.796;
   1:  PR[91,3] = PR[90,3] + 80.442;
   1:L PR[91] R[100]mm/sec CNT100;
   1:  PR[91,1] = PR[90,1] + 24.558;
   1:  PR[91,2] = PR[90,2] + 25.680;
   1:  PR[91,3] = PR[90,3] + 80.450;
   1:L PR[91] R[100]mm/sec CNT100;
   1:  PR[91,1] = PR[90,1] + 23.841;
   1:  PR[91,2] = PR[90,2] + 25.493;
   1:  PR[91,3] = PR[90,3] + 80.470;
   1:L PR[91] R[100]mm/sec CNT100;
   1:  PR[91,1] = PR[90,1] + 23.285;
   1:  PR[91,2] = PR[90,2] + 25.568;
   1:  PR[91,3] = PR[90,3] + 80.473;
   1:L PR[91] R[100]mm/sec CNT100;
   1:  PR[91,1] = PR[90,1] + 16.683;
   1:  PR[91,2] = PR[90,2] + 25.785;
   1:  PR[91,3] = PR[90,3] + 80.475;
   1:L PR[91] R[100]mm/sec CNT100;
   1:  PR[91,1] = PR[90,1] + 16.533;
   1:  PR[91,2] = PR[90,2] + 25.763;
   1:  PR[91,3] = PR[90,3] + 80.501;
   1:L PR[91] R[100]mm/sec CNT100;
   1:  PR[91,1] = PR[90,1] + 10.246;
   1:  PR[91,2] = PR[90,2] + 24.471;
   1:  PR[91,3] = PR[90,3] + 80.502;
   1:L PR[91] R[100]mm/sec CNT100;
   1:  PR[91,1] = PR[90,1] + 5.647;
   1:  PR[91,2] = PR[90,2] + 25.015;
   1:  PR[91,3] = PR[90,3] + 80.528;
   1:L PR[91] R[100]mm/sec CNT100;
   1:  PR[91,1] = PR[90,1] + 3.650;
   1:  PR[91,2] = PR[90,2] + 25.155;
   1:  PR[91,3] = PR[90,3] + 80.546;
   1:L PR[91] R[100]mm/sec CNT100;
   1:  PR[91,1] = PR[90,1] + 0.598;
   1:  PR[91,2] = PR[90,2] + 25.148;
   1:  PR[91,3] = PR[90,3] + 80.554;
   1:L PR[91] R[100]mm/sec CNT100;
   1:  PR[91,1] = PR[90,1] + -4.527;
   1:  PR[91,2] = PR[90,2] + 24.630;
   1:  PR[91,3] = PR[90,3] + 80.566;
   1:L PR[91] R[100]mm/sec CNT100;
   1:  PR[91,1] = PR[90,1] + -8.480;
   1:  PR[91,2] = PR[90,2] + 24.990;
   1:  PR[91,3] = PR[90,3] + 80.586;
   1:L PR[91] R[100]mm/sec CNT100;
   1:  PR[91,1] = PR[90,1] + -14.972;
   1:  PR[91,2] = PR[90,2] + 25.241;
   1:  PR[91,3] = PR[90,3] + 80.602;
   1:L PR[91] R[100]mm/sec CNT100;
   1:  PR[91,1] = PR[90,1] + -18.729;
   1:  PR[91,2] = PR[90,2] + 25.359;
   1:  PR[91,3] = PR[90,3] + 80.628;
   1:L PR[91] R[100]mm/sec CNT100;
   1:  PR[91,1] = PR[90,1] + -28.456;
   1:  PR[91,2] = PR[90,2] + 25.032;
   1:  PR[91,3] = PR[90,3] + 80.643;
   1:L PR[91] R[100]mm/sec CNT100;
   1:  PR[91,1] = PR[90,1] + -35.694;
   1:  PR[91,2] = PR[90,2] + 24.272;
   1:  PR[91,3] = PR[90,3] + 80.682;
   1:L PR[91] R[100]mm/sec CNT100;
   1:  PR[91,1] = PR[90,1] + -43.684;
   1:  PR[91,2] = PR[90,2] + 22.754;
   1:  PR[91,3] = PR[90,3] + 80.710;
   1:L PR[91] R[100]mm/sec CNT100;
   1:  PR[91,1] = PR[90,1] + -47.455;
   1:  PR[91,2] = PR[90,2] + 21.581;
   1:  PR[91,3] = PR[90,3] + 80.743;
   1:L PR[91] R[100]mm/sec CNT100;
   1:  PR[91,1] = PR[90,1] + -50.593;
   1:  PR[91,2] = PR[90,2] + 20.532;
   1:  PR[91,3] = PR[90,3] + 80.758;
   1:L PR[91] R[100]mm/sec CNT100;
   1:  PR[91,1] = PR[90,1] + -52.958;
   1:  PR[91,2] = PR[90,2] + 19.392;
   1:  PR[91,3] = PR[90,3] + 80.772;
   1:L PR[91] R[100]mm/sec CNT100;
   1:  PR[91,1] = PR[90,1] + -55.848;
   1:  PR[91,2] = PR[90,2] + 17.879;
   1:  PR[91,3] = PR[90,3] + 80.782;
   1:L PR[91] R[100]mm/sec CNT100;
   1:  PR[91] = PR[90];
   1:  PR[91,1] = PR[90,1] + -59.097;
   1:  PR[91,2] = PR[90,2] + 14.724;
   1:  PR[91,3] = PR[90,3] + 82.095;
   1:L PR[91] R[100]mm/sec CNT100;
   1:  PR[91,1] = PR[90,1] + -60.961;
   1:  PR[91,2] = PR[90,2] + 13.177;
   1:  PR[91,3] = PR[90,3] + 80.812;
   1:L PR[91] R[100]mm/sec CNT100;
   1:  PR[91,1] = PR[90,1] + -62.361;
   1:  PR[91,2] = PR[90,2] + 11.459;
   1:  PR[91,3] = PR[90,3] + 80.822;
   1:L PR[91] R[100]mm/sec CNT100;
   1:  PR[91,1] = PR[90,1] + -64.566;
   1:  PR[91,2] = PR[90,2] + 8.651;
   1:  PR[91,3] = PR[90,3] + 80.831;
   1:L PR[91] R[100]mm/sec CNT100;
   1:  PR[91,1] = PR[90,1] + -64.934;
   1:  PR[91,2] = PR[90,2] + 7.850;
   1:  PR[91,3] = PR[90,3] + 80.845;
   1:L PR[91] R[100]mm/sec CNT100;
   1:  PR[91,1] = PR[90,1] + -66.656;
   1:  PR[91,2] = PR[90,2] + 3.986;
   1:  PR[91,3] = PR[90,3] + 80.849;
   1:L PR[91] R[100]mm/sec CNT100;
   1:  PR[91,1] = PR[90,1] + -67.348;
   1:  PR[91,2] = PR[90,2] + -0.728;
   1:  PR[91,3] = PR[90,3] + 80.866;
   1:L PR[91] R[100]mm/sec CNT100;
   1:  PR[91,1] = PR[90,1] + -66.993;
   1:  PR[91,2] = PR[90,2] + -2.684;
   1:  PR[91,3] = PR[90,3] + 80.885;
   1:L PR[91] R[100]mm/sec CNT100;
   1:  PR[91,1] = PR[90,1] + -66.707;
   1:  PR[91,2] = PR[90,2] + -3.713;
   1:  PR[91,3] = PR[90,3] + 80.893;
   1:L PR[91] R[100]mm/sec CNT100;
   1:  PR[91,1] = PR[90,1] + -66.475;
   1:  PR[91,2] = PR[90,2] + -5.456;
   1:  PR[91,3] = PR[90,3] + 80.897;
   1:L PR[91] R[100]mm/sec CNT100;
   1:  PR[91,1] = PR[90,1] + -65.707;
   1:  PR[91,2] = PR[90,2] + -7.317;
   1:  PR[91,3] = PR[90,3] + 80.904;
   1:L PR[91] R[100]mm/sec CNT100;
   1:  PR[91,1] = PR[90,1] + -64.534;
   1:  PR[91,2] = PR[90,2] + -9.975;
   1:  PR[91,3] = PR[90,3] + 80.912;
   1:L PR[91] R[100]mm/sec CNT100;
   1:  PR[91,1] = PR[90,1] + -62.639;
   1:  PR[91,2] = PR[90,2] + -12.585;
   1:  PR[91,3] = PR[90,3] + 80.924;
   1:L PR[91] R[100]mm/sec CNT100;
   1:  PR[91,1] = PR[90,1] + -61.422;
   1:  PR[91,2] = PR[90,2] + -14.146;
   1:  PR[91,3] = PR[90,3] + 80.937;
   1:L PR[91] R[100]mm/sec CNT100;
   1:  PR[91,1] = PR[90,1] + -57.445;
   1:  PR[91,2] = PR[90,2] + -17.734;
   1:  PR[91,3] = PR[90,3] + 80.945;
   1:L PR[91] R[100]mm/sec CNT100;
   1:  PR[91,1] = PR[90,1] + -57.362;
   1:  PR[91,2] = PR[90,2] + -17.803;
   1:  PR[91,3] = PR[90,3] + 80.967;
   1:L PR[91] R[100]mm/sec CNT100;
   1:  PR[91,1] = PR[90,1] + -56.971;
   1:  PR[91,2] = PR[90,2] + -18.043;
   1:L PR[91] R[100]mm/sec CNT100;
   1:  PR[91,1] = PR[90,1] + -52.816;
   1:  PR[91,2] = PR[90,2] + -20.339;
   1:  PR[91,3] = PR[90,3] + 80.969;
   1:L PR[91] R[100]mm/sec CNT100;
   1:  PR[91,1] = PR[90,1] + -50.855;
   1:  PR[91,2] = PR[90,2] + -21.359;
   1:  PR[91,3] = PR[90,3] + 80.988;
   1:L PR[91] R[100]mm/sec CNT100;
   1:  PR[91,1] = PR[90,1] + -47.969;
   1:  PR[91,2] = PR[90,2] + -22.438;
   1:  PR[91,3] = PR[90,3] + 80.997;
   1:L PR[91] R[100]mm/sec CNT100;
   1:  PR[91,1] = PR[90,1] + -43.135;
   1:  PR[91,2] = PR[90,2] + -24.088;
   1:  PR[91,3] = PR[90,3] + 81.009;
   1:L PR[91] R[100]mm/sec CNT100;
   1:  PR[91,1] = PR[90,1] + -42.305;
   1:  PR[91,2] = PR[90,2] + -24.336;
   1:  PR[91,3] = PR[90,3] + 81.030;
   1:L PR[91] R[100]mm/sec CNT100;
   1:  PR[91,1] = PR[90,1] + -40.753;
   1:  PR[91,2] = PR[90,2] + -24.637;
   1:  PR[91,3] = PR[90,3] + 81.033;
   1:L PR[91] R[100]mm/sec CNT100;
   1:  PR[91,1] = PR[90,1] + -34.092;
   1:  PR[91,2] = PR[90,2] + -25.875;
   1:  PR[91,3] = PR[90,3] + 81.039;
   1:L PR[91] R[100]mm/sec CNT100;
   1:  PR[91,1] = PR[90,1] + -25.910;
   1:  PR[91,2] = PR[90,2] + -26.735;
   1:  PR[91,3] = PR[90,3] + 81.067;
   1:L PR[91] R[100]mm/sec CNT100;
   1:  PR[91,1] = PR[90,1] + -16.101;
   1:  PR[91,2] = PR[90,2] + -27.071;
   1:  PR[91,3] = PR[90,3] + 81.100;
   1:L PR[91] R[100]mm/sec CNT100;
   1:  PR[91,1] = PR[90,1] + -11.322;
   1:  PR[91,2] = PR[90,2] + -26.920;
   1:  PR[91,3] = PR[90,3] + 81.139;
   1:L PR[91] R[100]mm/sec CNT100;
   1:  PR[91,1] = PR[90,1] + -6.014;
   1:  PR[91,2] = PR[90,2] + -26.721;
   1:  PR[91,3] = PR[90,3] + 81.158;
   1:L PR[91] R[100]mm/sec CNT100;
   1:  PR[91,1] = PR[90,1] + -5.208;
   1:  PR[91,2] = PR[90,2] + -26.663;
   1:  PR[91,3] = PR[90,3] + 81.180;
   1:L PR[91] R[100]mm/sec CNT100;
   1:  PR[91,1] = PR[90,1] + -3.478;
   1:  PR[91,2] = PR[90,2] + -26.467;
   1:  PR[91,3] = PR[90,3] + 81.183;
   1:L PR[91] R[100]mm/sec CNT100;
   1:  PR[91,1] = PR[90,1] + -2.707;
   1:  PR[91,2] = PR[90,2] + -26.446;
   1:  PR[91,3] = PR[90,3] + 81.190;
   1:L PR[91] R[100]mm/sec CNT100;
   1:  PR[91,1] = PR[90,1] + 0.335;
   1:  PR[91,2] = PR[90,2] + -26.763;
   1:  PR[91,3] = PR[90,3] + 81.193;
   1:L PR[91] R[100]mm/sec CNT100;
   1:  PR[91,1] = PR[90,1] + 1.244;
   1:  PR[91,2] = PR[90,2] + -26.822;
   1:  PR[91,3] = PR[90,3] + 81.205;
   1:L PR[91] R[100]mm/sec CNT100;
   1:  PR[91,1] = PR[90,1] + 5.167;
   1:  PR[91,2] = PR[90,2] + -26.830;
   1:  PR[91,3] = PR[90,3] + 81.209;
   1:L PR[91] R[100]mm/sec CNT100;
   1:  PR[91,1] = PR[90,1] + 6.150;
   1:  PR[91,2] = PR[90,2] + -26.762;
   1:  PR[91,3] = PR[90,3] + 81.225;
   1:L PR[91] R[100]mm/sec CNT100;
   1:  PR[91,1] = PR[90,1] + 8.363;
   1:  PR[91,2] = PR[90,2] + -26.500;
   1:  PR[91,3] = PR[90,3] + 81.229;
   1:L PR[91] R[100]mm/sec CNT100;
   1:  PR[91,1] = PR[90,1] + 10.803;
   1:  PR[91,2] = PR[90,2] + -26.256;
   1:  PR[91,3] = PR[90,3] + 81.238;
   1:L PR[91] R[100]mm/sec CNT100;
   1:  PR[91,1] = PR[90,1] + 15.320;
   1:  PR[91,2] = PR[90,2] + -27.185;
   1:  PR[91,3] = PR[90,3] + 81.248;
   1:L PR[91] R[100]mm/sec CNT100;
   1:  PR[91,1] = PR[90,1] + 16.175;
   1:  PR[91,2] = PR[90,2] + -27.328;
   1:  PR[91,3] = PR[90,3] + 81.266;
   1:L PR[91] R[100]mm/sec CNT100;
   1:  PR[91,1] = PR[90,1] + 16.871;
   1:  PR[91,2] = PR[90,2] + -27.413;
   1:  PR[91,3] = PR[90,3] + 81.270;
   1:L PR[91] R[100]mm/sec CNT100;
   1:  PR[91,1] = PR[90,1] + 23.534;
   1:  PR[91,2] = PR[90,2] + -27.191;
   1:  PR[91,3] = PR[90,3] + 81.272;
   1:L PR[91] R[100]mm/sec CNT100;
   1:  PR[91,1] = PR[90,1] + 26.132;
   1:  PR[91,2] = PR[90,2] + -27.811;
   1:  PR[91,3] = PR[90,3] + 81.299;
   1:L PR[91] R[100]mm/sec CNT100;
   1:  PR[91,1] = PR[90,1] + 29.056;
   1:  PR[91,2] = PR[90,2] + -28.481;
   1:  PR[91,3] = PR[90,3] + 81.310;
   1:L PR[91] R[100]mm/sec CNT100;
   1:  PR[91,1] = PR[90,1] + 29.886;
   1:  PR[91,2] = PR[90,2] + -28.547;
   1:  PR[91,3] = PR[90,3] + 81.322;
   1:L PR[91] R[100]mm/sec CNT100;
   1:  PR[91,1] = PR[90,1] + 34.276;
   1:  PR[91,2] = PR[90,2] + -28.794;
   1:  PR[91,3] = PR[90,3] + 81.325;
   1:L PR[91] R[100]mm/sec CNT100;
   1:  PR[91,1] = PR[90,1] + 37.303;
   1:  PR[91,2] = PR[90,2] + -28.504;
   1:  PR[91,3] = PR[90,3] + 81.343;
   1:L PR[91] R[100]mm/sec CNT100;
   1:  PR[91,1] = PR[90,1] + 39.402;
   1:  PR[91,2] = PR[90,2] + -28.267;
   1:  PR[91,3] = PR[90,3] + 81.355;
   1:L PR[91] R[100]mm/sec CNT100;
   1:  PR[91,1] = PR[90,1] + 43.418;
   1:  PR[91,2] = PR[90,2] + -27.157;
   1:  PR[91,3] = PR[90,3] + 81.364;
   1:L PR[91] R[100]mm/sec CNT100;
   1:  PR[91,1] = PR[90,1] + 44.378;
   1:  PR[91,2] = PR[90,2] + -26.927;
   1:  PR[91,3] = PR[90,3] + 81.381;
   1:L PR[91] R[100]mm/sec CNT100;
   1:  PR[91,1] = PR[90,1] + 44.728;
   1:  PR[91,2] = PR[90,2] + -26.809;
   1:  PR[91,3] = PR[90,3] + 81.385;
   1:L PR[91] R[100]mm/sec CNT100;
   1:  PR[91,1] = PR[90,1] + 48.444;
   1:  PR[91,2] = PR[90,2] + -25.257;
   1:  PR[91,3] = PR[90,3] + 81.386;
   1:L PR[91] R[100]mm/sec CNT100;
   1:  PR[91,1] = PR[90,1] + 50.965;
   1:  PR[91,2] = PR[90,2] + -23.942;
   1:  PR[91,3] = PR[90,3] + 81.402;
   1:L PR[91] R[100]mm/sec CNT100;
   1:  PR[91,1] = PR[90,1] + 51.821;
   1:  PR[91,2] = PR[90,2] + -23.403;
   1:  PR[91,3] = PR[90,3] + 81.414;
   1:L PR[91] R[100]mm/sec CNT100;
   1:  PR[91,1] = PR[90,1] + 53.101;
   1:  PR[91,2] = PR[90,2] + -22.447;
   1:  PR[91,3] = PR[90,3] + 81.418;
   1:L PR[91] R[100]mm/sec CNT100;
   1:  PR[91,1] = PR[90,1] + 55.414;
   1:  PR[91,2] = PR[90,2] + -21.045;
   1:  PR[91,3] = PR[90,3] + 81.424;
   1:L PR[91] R[100]mm/sec CNT100;
   1:  PR[91,1] = PR[90,1] + 57.005;
   1:  PR[91,2] = PR[90,2] + -19.852;
   1:  PR[91,3] = PR[90,3] + 81.435;
   1:L PR[91] R[100]mm/sec CNT100;
   1:  PR[91,1] = PR[90,1] + 58.345;
   1:  PR[91,2] = PR[90,2] + -18.719;
   1:  PR[91,3] = PR[90,3] + 81.443;
   1:L PR[91] R[100]mm/sec CNT100;
   1:  PR[91,1] = PR[90,1] + 59.721;
   1:  PR[91,2] = PR[90,2] + -17.321;
   1:  PR[91,3] = PR[90,3] + 81.450;
   1:L PR[91] R[100]mm/sec CNT100;
   1:  PR[91,1] = PR[90,1] + 61.308;
   1:  PR[91,2] = PR[90,2] + -15.938;
   1:  PR[91,3] = PR[90,3] + 81.458;
   1:L PR[91] R[100]mm/sec CNT100;
   1:  PR[91,1] = PR[90,1] + 62.644;
   1:  PR[91,2] = PR[90,2] + -14.376;
   1:  PR[91,3] = PR[90,3] + 81.466;
   1:L PR[91] R[100]mm/sec CNT100;
   1:  PR[91,1] = PR[90,1] + 64.150;
   1:  PR[91,2] = PR[90,2] + -12.560;
   1:  PR[91,3] = PR[90,3] + 81.475;
   1:L PR[91] R[100]mm/sec CNT100;
   1:  PR[91,1] = PR[90,1] + 66.017;
   1:  PR[91,2] = PR[90,2] + -9.345;
   1:  PR[91,3] = PR[90,3] + 81.484;
   1:L PR[91] R[100]mm/sec CNT100;
   1:  PR[91,1] = PR[90,1] + 66.304;
   1:  PR[91,2] = PR[90,2] + -8.829;
   1:  PR[91,3] = PR[90,3] + 81.499;
   1:L PR[91] R[100]mm/sec CNT100;
   1:  PR[91,1] = PR[90,1] + 67.558;
   1:  PR[91,2] = PR[90,2] + -4.939;
   1:  PR[91,3] = PR[90,3] + 81.501;
   1:L PR[91] R[100]mm/sec CNT100;
   1:  PR[91,1] = PR[90,1] + 67.624;
   1:  PR[91,2] = PR[90,2] + -4.472;
   1:  PR[91,3] = PR[90,3] + 81.518;
   1:L PR[91] R[100]mm/sec CNT100;
   1:  PR[91,1] = PR[90,1] + 68.015;
   1:  PR[91,2] = PR[90,2] + -0.768;
   1:  PR[91,3] = PR[90,3] + 81.520;
   1:L PR[91] R[100]mm/sec CNT100;
   1:  PR[91,1] = PR[90,1] + 67.931;
   1:  PR[91,2] = PR[90,2] + -0.182;
   1:  PR[91,3] = PR[90,3] + 81.535;
   1:L PR[91] R[100]mm/sec CNT100;
   1:  PR[91,1] = PR[90,1] + 67.546;
   1:  PR[91,2] = PR[90,2] + 3.516;
   1:  PR[91,3] = PR[90,3] + 81.537;
   1:L PR[91] R[100]mm/sec CNT100;
   1:  PR[91,1] = PR[90,1] + 66.304;
   1:  PR[91,2] = PR[90,2] + 7.370;
   1:  PR[91,3] = PR[90,3] + 81.552;
   1:L PR[91] R[100]mm/sec CNT100;
   1:  PR[91,1] = PR[90,1] + 66.017;
   1:  PR[91,2] = PR[90,2] + 7.887;
   1:  PR[91,3] = PR[90,3] + 81.568;
   1:L PR[91] R[100]mm/sec CNT100;
   1:  PR[91,1] = PR[90,1] + 64.150;
   1:  PR[91,2] = PR[90,2] + 11.101;
   1:  PR[91,3] = PR[90,3] + 81.571;
   1:L PR[91] R[100]mm/sec CNT100;
   1:  PR[91,1] = PR[90,1] + 62.644;
   1:  PR[91,2] = PR[90,2] + 12.917;
   1:  PR[91,3] = PR[90,3] + 81.586;
   1:L PR[91] R[100]mm/sec CNT100;
   1:  PR[91,1] = PR[90,1] + 61.308;
   1:  PR[91,2] = PR[90,2] + 14.480;
   1:  PR[91,3] = PR[90,3] + 81.595;
   1:L PR[91] R[100]mm/sec CNT100;
   1:  PR[91,1] = PR[90,1] + 59.721;
   1:  PR[91,2] = PR[90,2] + 15.862;
   1:  PR[91,3] = PR[90,3] + 81.603;
   1:L PR[91] R[100]mm/sec CNT100;
   1:  PR[91,1] = PR[90,1] + 58.345;
   1:  PR[91,2] = PR[90,2] + 17.260;
   1:  PR[91,3] = PR[90,3] + 81.612;
   1:L PR[91] R[100]mm/sec CNT100;
   1:  PR[91,1] = PR[90,1] + 57.004;
   1:  PR[91,2] = PR[90,2] + 18.393;
   1:  PR[91,3] = PR[90,3] + 81.620;
   1:L PR[91] R[100]mm/sec CNT100;
   1:  PR[91,1] = PR[90,1] + 55.414;
   1:  PR[91,2] = PR[90,2] + 19.586;
   1:  PR[91,3] = PR[90,3] + 81.627;
   1:L PR[91] R[100]mm/sec CNT100;
   1:  PR[91,1] = PR[90,1] + 53.101;
   1:  PR[91,2] = PR[90,2] + 20.989;
   1:  PR[91,3] = PR[90,3] + 81.635;
   1:L PR[91] R[100]mm/sec CNT100;
   1:  PR[91,1] = PR[90,1] + 51.821;
   1:  PR[91,2] = PR[90,2] + 21.944;
   1:  PR[91,3] = PR[90,3] + 81.646;
   1:L PR[91] R[100]mm/sec CNT100;
   1:  PR[91,1] = PR[90,1] + 50.965;
   1:  PR[91,2] = PR[90,2] + 22.483;
   1:  PR[91,3] = PR[90,3] + 81.652;
   1:L PR[91] R[100]mm/sec CNT100;
   1:  PR[91,1] = PR[90,1] + 48.444;
   1:  PR[91,2] = PR[90,2] + 23.798;
   1:  PR[91,3] = PR[90,3] + 81.656;
   1:L PR[91] R[100]mm/sec CNT100;
   1:  PR[91,1] = PR[90,1] + 44.728;
   1:  PR[91,2] = PR[90,2] + 25.350;
   1:  PR[91,3] = PR[90,3] + 81.668;
   1:L PR[91] R[100]mm/sec CNT100;
   1:  PR[91,1] = PR[90,1] + 44.378;
   1:  PR[91,2] = PR[90,2] + 25.468;
   1:  PR[91,3] = PR[90,3] + 81.684;
   1:L PR[91] R[100]mm/sec CNT100;
   1:  PR[91,1] = PR[90,1] + 43.418;
   1:  PR[91,2] = PR[90,2] + 25.698;
   1:  PR[91,3] = PR[90,3] + 81.685;
   1:L PR[91] R[100]mm/sec CNT100;
   1:  PR[91,1] = PR[90,1] + 39.402;
   1:  PR[91,2] = PR[90,2] + 26.808;
   1:  PR[91,3] = PR[90,3] + 81.689;
   1:L PR[91] R[100]mm/sec CNT100;
   1:  PR[91,1] = PR[90,1] + 37.303;
   1:  PR[91,2] = PR[90,2] + 27.046;
   1:  PR[91,3] = PR[90,3] + 81.706;
   1:L PR[91] R[100]mm/sec CNT100;
   1:  PR[91,1] = PR[90,1] + 34.276;
   1:  PR[91,2] = PR[90,2] + 27.336;
   1:  PR[91,3] = PR[90,3] + 81.714;
   1:L PR[91] R[100]mm/sec CNT100;
   1:  PR[91,1] = PR[90,1] + 29.886;
   1:  PR[91,2] = PR[90,2] + 27.088;
   1:  PR[91,3] = PR[90,3] + 81.727;
   1:L PR[91] R[100]mm/sec CNT100;
   1:  PR[91,1] = PR[90,1] + 29.056;
   1:  PR[91,2] = PR[90,2] + 27.022;
   1:  PR[91,3] = PR[90,3] + 81.744;
   1:L PR[91] R[100]mm/sec CNT100;
   1:  PR[91,1] = PR[90,1] + 26.131;
   1:  PR[91,2] = PR[90,2] + 26.352;
   1:  PR[91,3] = PR[90,3] + 81.748;
   1:L PR[91] R[100]mm/sec CNT100;
   1:  PR[91,1] = PR[90,1] + 23.532;
   1:  PR[91,2] = PR[90,2] + 25.732;
   1:  PR[91,3] = PR[90,3] + 81.760;
   1:L PR[91] R[100]mm/sec CNT100;
   1:  PR[91,1] = PR[90,1] + 17.636;
   1:  PR[91,2] = PR[90,2] + 25.942;
   1:  PR[91,3] = PR[90,3] + 81.770;
   1:L PR[91] R[100]mm/sec CNT100;
   1:  PR[91,1] = PR[90,1] + 16.885;
   1:  PR[91,2] = PR[90,2] + 25.956;
   1:  PR[91,3] = PR[90,3] + 81.794;
   1:L PR[91] R[100]mm/sec CNT100;
   1:  PR[91,1] = PR[90,1] + 16.176;
   1:  PR[91,2] = PR[90,2] + 25.869;
   1:  PR[91,3] = PR[90,3] + 81.797;
   1:L PR[91] R[100]mm/sec CNT100;
   1:  PR[91,1] = PR[90,1] + 15.321;
   1:  PR[91,2] = PR[90,2] + 25.726;
   1:  PR[91,3] = PR[90,3] + 81.800;
   1:L PR[91] R[100]mm/sec CNT100;
   1:  PR[91,1] = PR[90,1] + 10.804;
   1:  PR[91,2] = PR[90,2] + 24.798;
   1:  PR[91,3] = PR[90,3] + 81.804;
   1:L PR[91] R[100]mm/sec CNT100;
   1:  PR[91,1] = PR[90,1] + 8.361;
   1:  PR[91,2] = PR[90,2] + 25.041;
   1:  PR[91,3] = PR[90,3] + 81.822;
   1:L PR[91] R[100]mm/sec CNT100;
   1:  PR[91,1] = PR[90,1] + 6.155;
   1:  PR[91,2] = PR[90,2] + 25.303;
   1:  PR[91,3] = PR[90,3] + 81.832;
   1:L PR[91] R[100]mm/sec CNT100;
   1:  PR[91,1] = PR[90,1] + 5.173;
   1:  PR[91,2] = PR[90,2] + 25.372;
   1:  PR[91,3] = PR[90,3] + 81.841;
   1:L PR[91] R[100]mm/sec CNT100;
   1:  PR[91,1] = PR[90,1] + 1.298;
   1:  PR[91,2] = PR[90,2] + 25.364;
   1:  PR[91,3] = PR[90,3] + 81.845;
   1:L PR[91] R[100]mm/sec CNT100;
   1:  PR[91,1] = PR[90,1] + -2.664;
   1:  PR[91,2] = PR[90,2] + 24.963;
   1:  PR[91,3] = PR[90,3] + 81.860;
   1:L PR[91] R[100]mm/sec CNT100;
   1:  PR[91,1] = PR[90,1] + -5.173;
   1:  PR[91,2] = PR[90,2] + 25.202;
   1:  PR[91,3] = PR[90,3] + 81.876;
   1:L PR[91] R[100]mm/sec CNT100;
   1:  PR[91,1] = PR[90,1] + -5.712;
   1:  PR[91,2] = PR[90,2] + 25.242;
   1:  PR[91,3] = PR[90,3] + 81.887;
   1:L PR[91] R[100]mm/sec CNT100;
   1:  PR[91,1] = PR[90,1] + -11.323;
   1:  PR[91,2] = PR[90,2] + 25.461;
   1:  PR[91,3] = PR[90,3] + 81.889;
   1:L PR[91] R[100]mm/sec CNT100;
   1:  PR[91,1] = PR[90,1] + -16.101;
   1:  PR[91,2] = PR[90,2] + 25.612;
   1:  PR[91,3] = PR[90,3] + 81.911;
   1:L PR[91] R[100]mm/sec CNT100;
   1:  PR[91,1] = PR[90,1] + -25.910;
   1:  PR[91,2] = PR[90,2] + 25.277;
   1:  PR[91,3] = PR[90,3] + 81.930;
   1:L PR[91] R[100]mm/sec CNT100;
   1:  PR[91,1] = PR[90,1] + -34.129;
   1:  PR[91,2] = PR[90,2] + 24.417;
   1:  PR[91,3] = PR[90,3] + 81.970;
   1:L PR[91] R[100]mm/sec CNT100;
   1:  PR[91,1] = PR[90,1] + -42.483;
   1:  PR[91,2] = PR[90,2] + 22.838;
   1:  PR[91,3] = PR[90,3] + 82.003;
   1:L PR[91] R[100]mm/sec CNT100;
   1:  PR[91,1] = PR[90,1] + -43.134;
   1:  PR[91,2] = PR[90,2] + 22.635;
   1:  PR[91,3] = PR[90,3] + 82.037;
   1:L PR[91] R[100]mm/sec CNT100;
   1:  PR[91,1] = PR[90,1] + -49.319;
   1:  PR[91,2] = PR[90,2] + 20.568;
   1:  PR[91,3] = PR[90,3] + 82.040;
   1:L PR[91] R[100]mm/sec CNT100;
   1:  PR[91,1] = PR[90,1] + -54.015;
   1:  PR[91,2] = PR[90,2] + 18.303;
   1:  PR[91,3] = PR[90,3] + 82.066;
   1:L PR[91] R[100]mm/sec CNT100;
   1:  PR[91,1] = PR[90,1] + -55.257;
   1:  PR[91,2] = PR[90,2] + 17.653;
   1:  PR[91,3] = PR[90,3] + 82.087;
   1:L PR[91] R[100]mm/sec CNT100;
   1:  PR[91,1] = PR[90,1] + -55.728;
   1:  PR[91,2] = PR[90,2] + 17.390;
   1:  PR[91,3] = PR[90,3] + 82.093;
   1:L PR[91] R[100]mm/sec CNT100;
   1:  PR[91] = PR[90];
   1:  PR[91,1] = PR[90,1] + -58.434;
   1:  PR[91,2] = PR[90,2] + 14.368;
   1:  PR[91,3] = PR[90,3] + 83.395;
   1:L PR[91] R[100]mm/sec CNT100;
   1:  PR[91,1] = PR[90,1] + -59.656;
   1:  PR[91,2] = PR[90,2] + 13.353;
   1:  PR[91,3] = PR[90,3] + 82.114;
   1:L PR[91] R[100]mm/sec CNT100;
   1:  PR[91,1] = PR[90,1] + -61.596;
   1:  PR[91,2] = PR[90,2] + 10.973;
   1:  PR[91,3] = PR[90,3] + 82.120;
   1:L PR[91] R[100]mm/sec CNT100;
   1:  PR[91,1] = PR[90,1] + -63.324;
   1:  PR[91,2] = PR[90,2] + 8.772;
   1:  PR[91,3] = PR[90,3] + 82.133;
   1:L PR[91] R[100]mm/sec CNT100;
   1:  PR[91,1] = PR[90,1] + -64.034;
   1:  PR[91,2] = PR[90,2] + 7.229;
   1:  PR[91,3] = PR[90,3] + 82.144;
   1:L PR[91] R[100]mm/sec CNT100;
   1:  PR[91,1] = PR[90,1] + -65.452;
   1:  PR[91,2] = PR[90,2] + 4.047;
   1:  PR[91,3] = PR[90,3] + 82.151;
   1:L PR[91] R[100]mm/sec CNT100;
   1:  PR[91,1] = PR[90,1] + -66.056;
   1:  PR[91,2] = PR[90,2] + -0.072;
   1:  PR[91,3] = PR[90,3] + 82.165;
   1:L PR[91] R[100]mm/sec CNT100;
   1:  PR[91,1] = PR[90,1] + -66.225;
   1:  PR[91,2] = PR[90,2] + -0.783;
   1:  PR[91,3] = PR[90,3] + 82.182;
   1:L PR[91] R[100]mm/sec CNT100;
   1:  PR[91,1] = PR[90,1] + -66.065;
   1:  PR[91,2] = PR[90,2] + -1.662;
   1:  PR[91,3] = PR[90,3] + 82.185;
   1:L PR[91] R[100]mm/sec CNT100;
   1:  PR[91,1] = PR[90,1] + -65.682;
   1:  PR[91,2] = PR[90,2] + -3.041;
   1:  PR[91,3] = PR[90,3] + 82.189;
   1:L PR[91] R[100]mm/sec CNT100;
   1:  PR[91,1] = PR[90,1] + -65.361;
   1:  PR[91,2] = PR[90,2] + -5.445;
   1:  PR[91,3] = PR[90,3] + 82.195;
   1:L PR[91] R[100]mm/sec CNT100;
   1:  PR[91,1] = PR[90,1] + -64.283;
   1:  PR[91,2] = PR[90,2] + -8.061;
   1:  PR[91,3] = PR[90,3] + 82.205;
   1:L PR[91] R[100]mm/sec CNT100;
   1:  PR[91,1] = PR[90,1] + -63.445;
   1:  PR[91,2] = PR[90,2] + -9.958;
   1:  PR[91,3] = PR[90,3] + 82.216;
   1:L PR[91] R[100]mm/sec CNT100;
   1:  PR[91,1] = PR[90,1] + -60.998;
   1:  PR[91,2] = PR[90,2] + -13.327;
   1:  PR[91,3] = PR[90,3] + 82.225;
   1:L PR[91] R[100]mm/sec CNT100;
   1:  PR[91,1] = PR[90,1] + -60.372;
   1:  PR[91,2] = PR[90,2] + -14.130;
   1:  PR[91,3] = PR[90,3] + 82.242;
   1:L PR[91] R[100]mm/sec CNT100;
   1:  PR[91,1] = PR[90,1] + -57.789;
   1:  PR[91,2] = PR[90,2] + -16.460;
   1:  PR[91,3] = PR[90,3] + 82.246;
   1:L PR[91] R[100]mm/sec CNT100;
   1:  PR[91,1] = PR[90,1] + -56.374;
   1:  PR[91,2] = PR[90,2] + -17.599;
   1:  PR[91,3] = PR[90,3] + 82.260;
   1:L PR[91] R[100]mm/sec CNT100;
   1:  PR[91,1] = PR[90,1] + -55.956;
   1:  PR[91,2] = PR[90,2] + -17.921;
   1:  PR[91,3] = PR[90,3] + 82.267;
   1:L PR[91] R[100]mm/sec CNT100;
   1:  PR[91,1] = PR[90,1] + -51.998;
   1:  PR[91,2] = PR[90,2] + -20.108;
   1:  PR[91,3] = PR[90,3] + 82.269;
   1:L PR[91] R[100]mm/sec CNT100;
   1:  PR[91,1] = PR[90,1] + -49.080;
   1:  PR[91,2] = PR[90,2] + -21.626;
   1:  PR[91,3] = PR[90,3] + 82.288;
   1:L PR[91] R[100]mm/sec CNT100;
   1:  PR[91,1] = PR[90,1] + -47.201;
   1:  PR[91,2] = PR[90,2] + -22.328;
   1:  PR[91,3] = PR[90,3] + 82.301;
   1:L PR[91] R[100]mm/sec CNT100;
   1:  PR[91,1] = PR[90,1] + -43.991;
   1:  PR[91,2] = PR[90,2] + -23.424;
   1:  PR[91,3] = PR[90,3] + 82.309;
   1:L PR[91] R[100]mm/sec CNT100;
   1:  PR[91,1] = PR[90,1] + -41.563;
   1:  PR[91,2] = PR[90,2] + -24.162;
   1:  PR[91,3] = PR[90,3] + 82.323;
   1:L PR[91] R[100]mm/sec CNT100;
   1:  PR[91,1] = PR[90,1] + -40.306;
   1:  PR[91,2] = PR[90,2] + -24.526;
   1:  PR[91,3] = PR[90,3] + 82.334;
   1:L PR[91] R[100]mm/sec CNT100;
   1:  PR[91,1] = PR[90,1] + -32.552;
   1:  PR[91,2] = PR[90,2] + -26.021;
   1:  PR[91,3] = PR[90,3] + 82.339;
   1:L PR[91] R[100]mm/sec CNT100;
   1:  PR[91,1] = PR[90,1] + -23.360;
   1:  PR[91,2] = PR[90,2] + -26.980;
   1:  PR[91,3] = PR[90,3] + 82.371;
   1:L PR[91] R[100]mm/sec CNT100;
   1:  PR[91,1] = PR[90,1] + -20.690;
   1:  PR[91,2] = PR[90,2] + -27.083;
   1:  PR[91,3] = PR[90,3] + 82.409;
   1:L PR[91] R[100]mm/sec CNT100;
   1:  PR[91,1] = PR[90,1] + -13.475;
   1:  PR[91,2] = PR[90,2] + -27.323;
   1:  PR[91,3] = PR[90,3] + 82.419;
   1:L PR[91] R[100]mm/sec CNT100;
   1:  PR[91,1] = PR[90,1] + -7.674;
   1:  PR[91,2] = PR[90,2] + -27.140;
   1:  PR[91,3] = PR[90,3] + 82.449;
   1:L PR[91] R[100]mm/sec CNT100;
   1:  PR[91,1] = PR[90,1] + -3.302;
   1:  PR[91,2] = PR[90,2] + -26.977;
   1:  PR[91,3] = PR[90,3] + 82.472;
   1:L PR[91] R[100]mm/sec CNT100;
   1:  PR[91,1] = PR[90,1] + -2.382;
   1:  PR[91,2] = PR[90,2] + -26.911;
   1:  PR[91,3] = PR[90,3] + 82.490;
   1:L PR[91] R[100]mm/sec CNT100;
   1:  PR[91,1] = PR[90,1] + -1.409;
   1:  PR[91,2] = PR[90,2] + -26.800;
   1:  PR[91,3] = PR[90,3] + 82.494;
   1:L PR[91] R[100]mm/sec CNT100;
   1:  PR[91,1] = PR[90,1] + -0.887;
   1:  PR[91,2] = PR[90,2] + -26.786;
   1:  PR[91,3] = PR[90,3] + 82.498;
   1:L PR[91] R[100]mm/sec CNT100;
   1:  PR[91,1] = PR[90,1] + 0.830;
   1:  PR[91,2] = PR[90,2] + -26.965;
   1:  PR[91,3] = PR[90,3] + 82.500;
   1:L PR[91] R[100]mm/sec CNT100;
   1:  PR[91,1] = PR[90,1] + 1.945;
   1:  PR[91,2] = PR[90,2] + -27.037;
   1:  PR[91,3] = PR[90,3] + 82.507;
   1:L PR[91] R[100]mm/sec CNT100;
   1:  PR[91,1] = PR[90,1] + 6.664;
   1:  PR[91,2] = PR[90,2] + -27.047;
   1:  PR[91,3] = PR[90,3] + 82.512;
   1:L PR[91] R[100]mm/sec CNT100;
   1:  PR[91,1] = PR[90,1] + 11.342;
   1:  PR[91,2] = PR[90,2] + -26.579;
   1:  PR[91,3] = PR[90,3] + 82.531;
   1:L PR[91] R[100]mm/sec CNT100;
   1:  PR[91,1] = PR[90,1] + 14.086;
   1:  PR[91,2] = PR[90,2] + -27.144;
   1:  PR[91,3] = PR[90,3] + 82.550;
   1:L PR[91] R[100]mm/sec CNT100;
   1:  PR[91,1] = PR[90,1] + 15.681;
   1:  PR[91,2] = PR[90,2] + -27.410;
   1:  PR[91,3] = PR[90,3] + 82.561;
   1:L PR[91] R[100]mm/sec CNT100;
   1:  PR[91,1] = PR[90,1] + 17.081;
   1:  PR[91,2] = PR[90,2] + -27.582;
   1:  PR[91,3] = PR[90,3] + 82.568;
   1:L PR[91] R[100]mm/sec CNT100;
   1:  PR[91,1] = PR[90,1] + 21.770;
   1:  PR[91,2] = PR[90,2] + -27.421;
   1:  PR[91,3] = PR[90,3] + 82.574;
   1:L PR[91] R[100]mm/sec CNT100;
   1:  PR[91,1] = PR[90,1] + 23.238;
   1:  PR[91,2] = PR[90,2] + -27.394;
   1:  PR[91,3] = PR[90,3] + 82.593;
   1:L PR[91] R[100]mm/sec CNT100;
   1:  PR[91,1] = PR[90,1] + 28.693;
   1:  PR[91,2] = PR[90,2] + -28.697;
   1:  PR[91,3] = PR[90,3] + 82.599;
   1:L PR[91] R[100]mm/sec CNT100;
   1:  PR[91,1] = PR[90,1] + 33.940;
   1:  PR[91,2] = PR[90,2] + -28.994;
   1:  PR[91,3] = PR[90,3] + 82.622;
   1:L PR[91] R[100]mm/sec CNT100;
   1:  PR[91,1] = PR[90,1] + 35.567;
   1:  PR[91,2] = PR[90,2] + -28.838;
   1:  PR[91,3] = PR[90,3] + 82.643;
   1:L PR[91] R[100]mm/sec CNT100;
   1:  PR[91,1] = PR[90,1] + 39.097;
   1:  PR[91,2] = PR[90,2] + -28.439;
   1:  PR[91,3] = PR[90,3] + 82.650;
   1:L PR[91] R[100]mm/sec CNT100;
   1:  PR[91,1] = PR[90,1] + 44.014;
   1:  PR[91,2] = PR[90,2] + -27.069;
   1:  PR[91,3] = PR[90,3] + 82.664;
   1:L PR[91] R[100]mm/sec CNT100;
   1:  PR[91,1] = PR[90,1] + 45.411;
   1:  PR[91,2] = PR[90,2] + -26.404;
   1:  PR[91,3] = PR[90,3] + 82.685;
   1:L PR[91] R[100]mm/sec CNT100;
   1:  PR[91,1] = PR[90,1] + 48.413;
   1:  PR[91,2] = PR[90,2] + -25.150;
   1:  PR[91,3] = PR[90,3] + 82.691;
   1:L PR[91] R[100]mm/sec CNT100;
   1:  PR[91,1] = PR[90,1] + 49.771;
   1:  PR[91,2] = PR[90,2] + -24.441;
   1:  PR[91,3] = PR[90,3] + 82.704;
   1:L PR[91] R[100]mm/sec CNT100;
   1:  PR[91,1] = PR[90,1] + 51.872;
   1:  PR[91,2] = PR[90,2] + -23.119;
   1:  PR[91,3] = PR[90,3] + 82.711;
   1:L PR[91] R[100]mm/sec CNT100;
   1:  PR[91,1] = PR[90,1] + 54.743;
   1:  PR[91,2] = PR[90,2] + -20.976;
   1:  PR[91,3] = PR[90,3] + 82.721;
   1:L PR[91] R[100]mm/sec CNT100;
   1:  PR[91,1] = PR[90,1] + 55.025;
   1:  PR[91,2] = PR[90,2] + -20.805;
   1:  PR[91,3] = PR[90,3] + 82.735;
   1:L PR[91] R[100]mm/sec CNT100;
   1:  PR[91,1] = PR[90,1] + 55.110;
   1:  PR[91,2] = PR[90,2] + -20.741;
   1:  PR[91,3] = PR[90,3] + 82.737;
   1:L PR[91] R[100]mm/sec CNT100;
   1:  PR[91,1] = PR[90,1] + 58.032;
   1:  PR[91,2] = PR[90,2] + -18.269;
   1:L PR[91] R[100]mm/sec CNT100;
   1:  PR[91,1] = PR[90,1] + 60.135;
   1:  PR[91,2] = PR[90,2] + -16.134;
   1:  PR[91,3] = PR[90,3] + 82.753;
   1:L PR[91] R[100]mm/sec CNT100;
   1:  PR[91,1] = PR[90,1] + 60.343;
   1:  PR[91,2] = PR[90,2] + -15.885;
   1:  PR[91,3] = PR[90,3] + 82.765;
   1:L PR[91] R[100]mm/sec CNT100;
   1:  PR[91,1] = PR[90,1] + 60.701;
   1:  PR[91,2] = PR[90,2] + -15.382;
   1:  PR[91,3] = PR[90,3] + 82.766;
   1:L PR[91] R[100]mm/sec CNT100;
   1:  PR[91,1] = PR[90,1] + 63.112;
   1:  PR[91,2] = PR[90,2] + -12.476;
   1:  PR[91,3] = PR[90,3] + 82.769;
   1:L PR[91] R[100]mm/sec CNT100;
   1:  PR[91,1] = PR[90,1] + 64.370;
   1:  PR[91,2] = PR[90,2] + -10.310;
   1:  PR[91,3] = PR[90,3] + 82.784;
   1:L PR[91] R[100]mm/sec CNT100;
   1:  PR[91,1] = PR[90,1] + 65.235;
   1:  PR[91,2] = PR[90,2] + -8.772;
   1:  PR[91,3] = PR[90,3] + 82.794;
   1:L PR[91] R[100]mm/sec CNT100;
   1:  PR[91,1] = PR[90,1] + 66.569;
   1:  PR[91,2] = PR[90,2] + -4.806;
   1:  PR[91,3] = PR[90,3] + 82.801;
   1:L PR[91] R[100]mm/sec CNT100;
   1:  PR[91,1] = PR[90,1] + 67.020;
   1:  PR[91,2] = PR[90,2] + -0.729;
   1:  PR[91,3] = PR[90,3] + 82.818;
   1:L PR[91] R[100]mm/sec CNT100;
   1:  PR[91,1] = PR[90,1] + 66.569;
   1:  PR[91,2] = PR[90,2] + 3.347;
   1:  PR[91,3] = PR[90,3] + 82.835;
   1:L PR[91] R[100]mm/sec CNT100;
   1:  PR[91,1] = PR[90,1] + 65.235;
   1:  PR[91,2] = PR[90,2] + 7.313;
   1:  PR[91,3] = PR[90,3] + 82.852;
   1:L PR[91] R[100]mm/sec CNT100;
   1:  PR[91,1] = PR[90,1] + 64.370;
   1:  PR[91,2] = PR[90,2] + 8.852;
   1:  PR[91,3] = PR[90,3] + 82.869;
   1:L PR[91] R[100]mm/sec CNT100;
   1:  PR[91,1] = PR[90,1] + 63.112;
   1:  PR[91,2] = PR[90,2] + 11.017;
   1:  PR[91,3] = PR[90,3] + 82.876;
   1:L PR[91] R[100]mm/sec CNT100;
   1:  PR[91,1] = PR[90,1] + 60.701;
   1:  PR[91,2] = PR[90,2] + 13.923;
   1:  PR[91,3] = PR[90,3] + 82.886;
   1:L PR[91] R[100]mm/sec CNT100;
   1:  PR[91,1] = PR[90,1] + 60.343;
   1:  PR[91,2] = PR[90,2] + 14.427;
   1:  PR[91,3] = PR[90,3] + 82.902;
   1:L PR[91] R[100]mm/sec CNT100;
   1:  PR[91,1] = PR[90,1] + 60.135;
   1:  PR[91,2] = PR[90,2] + 14.675;
   1:  PR[91,3] = PR[90,3] + 82.904;
   1:L PR[91] R[100]mm/sec CNT100;
   1:  PR[91,1] = PR[90,1] + 58.032;
   1:  PR[91,2] = PR[90,2] + 16.811;
   1:  PR[91,3] = PR[90,3] + 82.905;
   1:L PR[91] R[100]mm/sec CNT100;
   1:  PR[91,1] = PR[90,1] + 55.110;
   1:  PR[91,2] = PR[90,2] + 19.282;
   1:  PR[91,3] = PR[90,3] + 82.918;
   1:L PR[91] R[100]mm/sec CNT100;
   1:  PR[91,1] = PR[90,1] + 55.025;
   1:  PR[91,2] = PR[90,2] + 19.346;
   1:  PR[91,3] = PR[90,3] + 82.933;
   1:L PR[91] R[100]mm/sec CNT100;
   1:  PR[91,1] = PR[90,1] + 54.743;
   1:  PR[91,2] = PR[90,2] + 19.517;
   1:  PR[91,3] = PR[90,3] + 82.934;
   1:L PR[91] R[100]mm/sec CNT100;
   1:  PR[91,1] = PR[90,1] + 51.872;
   1:  PR[91,2] = PR[90,2] + 21.660;
   1:  PR[91,3] = PR[90,3] + 82.935;
   1:L PR[91] R[100]mm/sec CNT100;
   1:  PR[91,1] = PR[90,1] + 49.772;
   1:  PR[91,2] = PR[90,2] + 22.983;
   1:  PR[91,3] = PR[90,3] + 82.950;
   1:L PR[91] R[100]mm/sec CNT100;
   1:  PR[91,1] = PR[90,1] + 48.413;
   1:  PR[91,2] = PR[90,2] + 23.691;
   1:  PR[91,3] = PR[90,3] + 82.960;
   1:L PR[91] R[100]mm/sec CNT100;
   1:  PR[91,1] = PR[90,1] + 45.411;
   1:  PR[91,2] = PR[90,2] + 24.945;
   1:  PR[91,3] = PR[90,3] + 82.966;
   1:L PR[91] R[100]mm/sec CNT100;
   1:  PR[91,1] = PR[90,1] + 44.014;
   1:  PR[91,2] = PR[90,2] + 25.611;
   1:  PR[91,3] = PR[90,3] + 82.979;
   1:L PR[91] R[100]mm/sec CNT100;
   1:  PR[91,1] = PR[90,1] + 39.097;
   1:  PR[91,2] = PR[90,2] + 26.980;
   1:  PR[91,3] = PR[90,3] + 82.985;
   1:L PR[91] R[100]mm/sec CNT100;
   1:  PR[91,1] = PR[90,1] + 35.567;
   1:  PR[91,2] = PR[90,2] + 27.379;
   1:  PR[91,3] = PR[90,3] + 83.006;
   1:L PR[91] R[100]mm/sec CNT100;
   1:  PR[91,1] = PR[90,1] + 33.940;
   1:  PR[91,2] = PR[90,2] + 27.535;
   1:  PR[91,3] = PR[90,3] + 83.021;
   1:L PR[91] R[100]mm/sec CNT100;
   1:  PR[91,1] = PR[90,1] + 28.693;
   1:  PR[91,2] = PR[90,2] + 27.238;
   1:  PR[91,3] = PR[90,3] + 83.027;
   1:L PR[91] R[100]mm/sec CNT100;
   1:  PR[91,1] = PR[90,1] + 23.221;
   1:  PR[91,2] = PR[90,2] + 25.931;
   1:  PR[91,3] = PR[90,3] + 83.049;
   1:L PR[91] R[100]mm/sec CNT100;
   1:  PR[91,1] = PR[90,1] + 18.564;
   1:  PR[91,2] = PR[90,2] + 26.097;
   1:  PR[91,3] = PR[90,3] + 83.072;
   1:L PR[91] R[100]mm/sec CNT100;
   1:  PR[91,1] = PR[90,1] + 17.097;
   1:  PR[91,2] = PR[90,2] + 26.125;
   1:  PR[91,3] = PR[90,3] + 83.090;
   1:L PR[91] R[100]mm/sec CNT100;
   1:  PR[91,1] = PR[90,1] + 15.682;
   1:  PR[91,2] = PR[90,2] + 25.951;
   1:  PR[91,3] = PR[90,3] + 83.096;
   1:L PR[91] R[100]mm/sec CNT100;
   1:  PR[91,1] = PR[90,1] + 14.088;
   1:  PR[91,2] = PR[90,2] + 25.685;
   1:  PR[91,3] = PR[90,3] + 83.102;
   1:L PR[91] R[100]mm/sec CNT100;
   1:  PR[91,1] = PR[90,1] + 11.342;
   1:  PR[91,2] = PR[90,2] + 25.121;
   1:  PR[91,3] = PR[90,3] + 83.109;
   1:L PR[91] R[100]mm/sec CNT100;
   1:  PR[91,1] = PR[90,1] + 6.666;
   1:  PR[91,2] = PR[90,2] + 25.588;
   1:  PR[91,3] = PR[90,3] + 83.120;
   1:L PR[91] R[100]mm/sec CNT100;
   1:  PR[91,1] = PR[90,1] + 1.997;
   1:  PR[91,2] = PR[90,2] + 25.579;
   1:  PR[91,3] = PR[90,3] + 83.139;
   1:L PR[91] R[100]mm/sec CNT100;
   1:  PR[91,1] = PR[90,1] + -0.802;
   1:  PR[91,2] = PR[90,2] + 25.296;
   1:  PR[91,3] = PR[90,3] + 83.158;
   1:L PR[91] R[100]mm/sec CNT100;
   1:  PR[91,1] = PR[90,1] + -2.349;
   1:  PR[91,2] = PR[90,2] + 25.449;
   1:  PR[91,3] = PR[90,3] + 83.170;
   1:L PR[91] R[100]mm/sec CNT100;
   1:  PR[91,1] = PR[90,1] + -2.961;
   1:  PR[91,2] = PR[90,2] + 25.495;
   1:  PR[91,3] = PR[90,3] + 83.176;
   1:L PR[91] R[100]mm/sec CNT100;
   1:  PR[91,1] = PR[90,1] + -7.677;
   1:  PR[91,2] = PR[90,2] + 25.682;
   1:  PR[91,3] = PR[90,3] + 83.179;
   1:L PR[91] R[100]mm/sec CNT100;
   1:  PR[91,1] = PR[90,1] + -13.475;
   1:  PR[91,2] = PR[90,2] + 25.864;
   1:  PR[91,3] = PR[90,3] + 83.198;
   1:L PR[91] R[100]mm/sec CNT100;
   1:  PR[91,1] = PR[90,1] + -20.690;
   1:  PR[91,2] = PR[90,2] + 25.625;
   1:  PR[91,3] = PR[90,3] + 83.221;
   1:L PR[91] R[100]mm/sec CNT100;
   1:  PR[91,1] = PR[90,1] + -23.361;
   1:  PR[91,2] = PR[90,2] + 25.522;
   1:  PR[91,3] = PR[90,3] + 83.251;
   1:L PR[91] R[100]mm/sec CNT100;
   1:  PR[91,1] = PR[90,1] + -32.560;
   1:  PR[91,2] = PR[90,2] + 24.562;
   1:  PR[91,3] = PR[90,3] + 83.262;
   1:L PR[91] R[100]mm/sec CNT100;
   1:  PR[91,1] = PR[90,1] + -40.611;
   1:  PR[91,2] = PR[90,2] + 23.015;
   1:  PR[91,3] = PR[90,3] + 83.299;
   1:L PR[91] R[100]mm/sec CNT100;
   1:  PR[91,1] = PR[90,1] + -42.689;
   1:  PR[91,2] = PR[90,2] + 22.394;
   1:  PR[91,3] = PR[90,3] + 83.333;
   1:L PR[91] R[100]mm/sec CNT100;
   1:  PR[91,1] = PR[90,1] + -48.045;
   1:  PR[91,2] = PR[90,2] + 20.603;
   1:  PR[91,3] = PR[90,3] + 83.341;
   1:L PR[91] R[100]mm/sec CNT100;
   1:  PR[91,1] = PR[90,1] + -54.080;
   1:  PR[91,2] = PR[90,2] + 17.693;
   1:  PR[91,3] = PR[90,3] + 83.364;
   1:L PR[91] R[100]mm/sec CNT100;
   1:  PR[91,1] = PR[90,1] + -54.415;
   1:  PR[91,2] = PR[90,2] + 17.523;
   1:  PR[91,3] = PR[90,3] + 83.392;
   1:L PR[91] R[100]mm/sec CNT100;
   1:  PR[91,1] = PR[90,1] + -54.765;
   1:  PR[91,2] = PR[90,2] + 17.271;
   1:  PR[91,3] = PR[90,3] + 83.393;
   1:L PR[91] R[100]mm/sec CNT100;
   1:  PR[91] = PR[90];
   1:  PR[91,1] = PR[90,1] + -55.820;
   1:  PR[91,2] = PR[90,2] + 15.555;
   1:  PR[91,3] = PR[90,3] + 84.695;
   1:L PR[91] R[100]mm/sec CNT100;
   1:  PR[91,1] = PR[90,1] + -57.770;
   1:  PR[91,2] = PR[90,2] + 14.012;
   1:  PR[91,3] = PR[90,3] + 83.409;
   1:L PR[91] R[100]mm/sec CNT100;
   1:  PR[91,1] = PR[90,1] + -58.351;
   1:  PR[91,2] = PR[90,2] + 13.530;
   1:  PR[91,3] = PR[90,3] + 83.419;
   1:L PR[91] R[100]mm/sec CNT100;
   1:  PR[91,1] = PR[90,1] + -60.832;
   1:  PR[91,2] = PR[90,2] + 10.486;
   1:  PR[91,3] = PR[90,3] + 83.422;
   1:L PR[91] R[100]mm/sec CNT100;
   1:  PR[91,1] = PR[90,1] + -62.083;
   1:  PR[91,2] = PR[90,2] + 8.894;
   1:  PR[91,3] = PR[90,3] + 83.438;
   1:L PR[91] R[100]mm/sec CNT100;
   1:  PR[91,1] = PR[90,1] + -63.133;
   1:  PR[91,2] = PR[90,2] + 6.610;
   1:  PR[91,3] = PR[90,3] + 83.447;
   1:L PR[91] R[100]mm/sec CNT100;
   1:  PR[91,1] = PR[90,1] + -64.247;
   1:  PR[91,2] = PR[90,2] + 4.109;
   1:  PR[91,3] = PR[90,3] + 83.457;
   1:L PR[91] R[100]mm/sec CNT100;
   1:  PR[91,1] = PR[90,1] + -64.727;
   1:  PR[91,2] = PR[90,2] + 0.842;
   1:  PR[91,3] = PR[90,3] + 83.468;
   1:L PR[91] R[100]mm/sec CNT100;
   1:  PR[91,1] = PR[90,1] + -65.104;
   1:  PR[91,2] = PR[90,2] + -0.756;
   1:  PR[91,3] = PR[90,3] + 83.482;
   1:L PR[91] R[100]mm/sec CNT100;
   1:  PR[91,1] = PR[90,1] + -64.656;
   1:  PR[91,2] = PR[90,2] + -2.368;
   1:  PR[91,3] = PR[90,3] + 83.489;
   1:L PR[91] R[100]mm/sec CNT100;
   1:  PR[91,1] = PR[90,1] + -64.248;
   1:  PR[91,2] = PR[90,2] + -5.434;
